(* IEC 61131-3 sources: verifaps-lib/share/oscat, 100 files *)

(* ---- 10_standard.st ---- *)
// Down Counter

PROGRAM standard
  VAR_INPUT
    input : INT;
  END_VAR
  VAR
    reset, cnt, max, init : INT;
  END_VAR

  ACTION act_Init
    cnt := max;
  END_ACTION

  ACTION act_Check
  END_ACTION

  ACTION act_Count
    cnt := cnt - 1;
  END_ACTION

  ACTION act_Reset
    cnt := max;
  END_ACTION

  ACTION act_End
  END_ACTION

  INITIAL_STEP Init
    : act_Init(N);
  END_STEP

  STEP Check
    : act_Check(N);
  END_STEP

  STEP Count
    : act_Count(N);
  END_STEP

  STEP Reset
    : act_Reset(N);
  END_STEP

  STEP End
    : act_End(N);
  END_STEP

  TRANSITION FROM Init TO Check
    := init;
  END_TRANSITION
  TRANSITION FROM Check TO Count
    := input == 1 and cnt > 0;
  END_TRANSITION
  TRANSITION FROM Count TO Check
    := True;
  END_TRANSITION
  TRANSITION FROM Check TO Reset
    := reset == 1;
  END_TRANSITION
  TRANSITION FROM Reset TO Check
    := True;
  END_TRANSITION
END_PROGRAM

(* ---- 10_upgraded.st ---- *)
// Down Counter (Upgraded)

PROGRAM upgraded
  VAR_INPUT
    input : INT;
  END_VAR
  VAR
    reset, cnt, max, init : INT;
  END_VAR

  ACTION act_Init
    cnt := max;
  END_ACTION

  ACTION act_Check
  END_ACTION

  ACTION act_Count
    cnt := cnt - 2;
  END_ACTION

  ACTION act_Reset
    cnt := max;
  END_ACTION

  ACTION act_End
  END_ACTION

  INITIAL_STEP Init
    : act_Init(N);
  END_STEP

  STEP Check
    : act_Check(N);
  END_STEP

  STEP Count
    : act_Count(N);
  END_STEP

  STEP Reset
    : act_Reset(N);
  END_STEP

  STEP End
    : act_End(N);
  END_STEP

  TRANSITION FROM Init TO Check
    := init;
  END_TRANSITION
  TRANSITION FROM Check TO Count
    := input == 1 and cnt > 0;
  END_TRANSITION
  TRANSITION FROM Count TO Check
    := True;
  END_TRANSITION
  TRANSITION FROM Check TO Reset
    := reset == 1;
  END_TRANSITION
  TRANSITION FROM Reset TO Check
    := True;
  END_TRANSITION
END_PROGRAM

(* ---- 11_standard.st ---- *)
// Comparator Greater

PROGRAM standard
  VAR
    a, b, out, init : INT;
  END_VAR

  ACTION act_Init
    out := 0;
  END_ACTION

  ACTION act_Check
  END_ACTION

  ACTION act_Set
    out := 1;
  END_ACTION

  ACTION act_Reset
    out := 0;
  END_ACTION

  ACTION act_End
  END_ACTION

  INITIAL_STEP Init
    : act_Init(N);
  END_STEP

  STEP Check
    : act_Check(N);
  END_STEP

  STEP Set
    : act_Set(N);
  END_STEP

  STEP Reset
    : act_Reset(N);
  END_STEP

  STEP End
    : act_End(N);
  END_STEP

  TRANSITION FROM Init TO Check
    := init;
  END_TRANSITION
  TRANSITION FROM Check TO Set
    := a > b;
  END_TRANSITION
  TRANSITION FROM Check TO Reset
    := a <= b;
  END_TRANSITION
  TRANSITION FROM Set TO End
    := True;
  END_TRANSITION
  TRANSITION FROM Reset TO End
    := True;
  END_TRANSITION
END_PROGRAM

(* ---- 11_upgraded.st ---- *)
// Comparator Greater (Upgraded)

PROGRAM upgraded
  VAR
    a, b, out, init : INT;
  END_VAR

  ACTION act_Init
    out := 0;
  END_ACTION

  ACTION act_Check
  END_ACTION

  ACTION act_Set
    out := a - b;
  END_ACTION

  ACTION act_Reset
    out := 0;
  END_ACTION

  ACTION act_End
  END_ACTION

  INITIAL_STEP Init
    : act_Init(N);
  END_STEP

  STEP Check
    : act_Check(N);
  END_STEP

  STEP Set
    : act_Set(N);
  END_STEP

  STEP Reset
    : act_Reset(N);
  END_STEP

  STEP End
    : act_End(N);
  END_STEP

  TRANSITION FROM Init TO Check
    := init;
  END_TRANSITION
  TRANSITION FROM Check TO Set
    := a > b;
  END_TRANSITION
  TRANSITION FROM Check TO Reset
    := a <= b;
  END_TRANSITION
  TRANSITION FROM Set TO End
    := True;
  END_TRANSITION
  TRANSITION FROM Reset TO End
    := True;
  END_TRANSITION
END_PROGRAM

(* ---- 12_standard.st ---- *)
// Comparator Less

PROGRAM standard
  VAR
    a, b, out, init : INT;
  END_VAR

  ACTION act_Init
    out := 0;
  END_ACTION

  ACTION act_Check
  END_ACTION

  ACTION act_Set
    out := 1;
  END_ACTION

  ACTION act_Reset
    out := 0;
  END_ACTION

  ACTION act_End
  END_ACTION

  INITIAL_STEP Init
    : act_Init(N);
  END_STEP

  STEP Check
    : act_Check(N);
  END_STEP

  STEP Set
    : act_Set(N);
  END_STEP

  STEP Reset
    : act_Reset(N);
  END_STEP

  STEP End
    : act_End(N);
  END_STEP

  TRANSITION FROM Init TO Check
    := init;
  END_TRANSITION
  TRANSITION FROM Check TO Set
    := a < b;
  END_TRANSITION
  TRANSITION FROM Check TO Reset
    := a >= b;
  END_TRANSITION
  TRANSITION FROM Set TO End
    := True;
  END_TRANSITION
  TRANSITION FROM Reset TO End
    := True;
  END_TRANSITION
END_PROGRAM

(* ---- 12_upgraded.st ---- *)
// Comparator Less (Upgraded)

PROGRAM upgraded
  VAR
    a, b, out, init : INT;
  END_VAR

  ACTION act_Init
    out := 0;
  END_ACTION

  ACTION act_Check
  END_ACTION

  ACTION act_Set
    out := b - a;
  END_ACTION

  ACTION act_Reset
    out := 0;
  END_ACTION

  ACTION act_End
  END_ACTION

  INITIAL_STEP Init
    : act_Init(N);
  END_STEP

  STEP Check
    : act_Check(N);
  END_STEP

  STEP Set
    : act_Set(N);
  END_STEP

  STEP Reset
    : act_Reset(N);
  END_STEP

  STEP End
    : act_End(N);
  END_STEP

  TRANSITION FROM Init TO Check
    := init;
  END_TRANSITION
  TRANSITION FROM Check TO Set
    := a < b;
  END_TRANSITION
  TRANSITION FROM Check TO Reset
    := a >= b;
  END_TRANSITION
  TRANSITION FROM Set TO End
    := True;
  END_TRANSITION
  TRANSITION FROM Reset TO End
    := True;
  END_TRANSITION
END_PROGRAM

(* ---- 13_standard.st ---- *)
// Comparator Equal

PROGRAM standard
  VAR
    a, b, out, init : INT;
  END_VAR

  ACTION act_Init
    out := 0;
  END_ACTION

  ACTION act_Check
  END_ACTION

  ACTION act_Set
    out := 1;
  END_ACTION

  ACTION act_Reset
    out := 0;
  END_ACTION

  ACTION act_End
  END_ACTION

  INITIAL_STEP Init
    : act_Init(N);
  END_STEP

  STEP Check
    : act_Check(N);
  END_STEP

  STEP Set
    : act_Set(N);
  END_STEP

  STEP Reset
    : act_Reset(N);
  END_STEP

  STEP End
    : act_End(N);
  END_STEP

  TRANSITION FROM Init TO Check
    := init;
  END_TRANSITION
  TRANSITION FROM Check TO Set
    := a == b;
  END_TRANSITION
  TRANSITION FROM Check TO Reset
    := a != b;
  END_TRANSITION
  TRANSITION FROM Set TO End
    := True;
  END_TRANSITION
  TRANSITION FROM Reset TO End
    := True;
  END_TRANSITION
END_PROGRAM

(* ---- 13_upgraded.st ---- *)
// Comparator Equal (Upgraded)

PROGRAM upgraded
  VAR
    a, b, out, init : INT;
  END_VAR

  ACTION act_Init
    out := 0;
  END_ACTION

  ACTION act_Check
  END_ACTION

  ACTION act_Set
    out := a + b;
  END_ACTION

  ACTION act_Reset
    out := 0;
  END_ACTION

  ACTION act_End
  END_ACTION

  INITIAL_STEP Init
    : act_Init(N);
  END_STEP

  STEP Check
    : act_Check(N);
  END_STEP

  STEP Set
    : act_Set(N);
  END_STEP

  STEP Reset
    : act_Reset(N);
  END_STEP

  STEP End
    : act_End(N);
  END_STEP

  TRANSITION FROM Init TO Check
    := init;
  END_TRANSITION
  TRANSITION FROM Check TO Set
    := a == b;
  END_TRANSITION
  TRANSITION FROM Check TO Reset
    := a != b;
  END_TRANSITION
  TRANSITION FROM Set TO End
    := True;
  END_TRANSITION
  TRANSITION FROM Reset TO End
    := True;
  END_TRANSITION
END_PROGRAM

(* ---- 14_standard.st ---- *)
// Comparator Not Equal

PROGRAM standard
  VAR
    a, b, out, init : INT;
  END_VAR

  ACTION act_Init
    out := 0;
  END_ACTION

  ACTION act_Check
  END_ACTION

  ACTION act_Set
    out := 1;
  END_ACTION

  ACTION act_Reset
    out := 0;
  END_ACTION

  ACTION act_End
  END_ACTION

  INITIAL_STEP Init
    : act_Init(N);
  END_STEP

  STEP Check
    : act_Check(N);
  END_STEP

  STEP Set
    : act_Set(N);
  END_STEP

  STEP Reset
    : act_Reset(N);
  END_STEP

  STEP End
    : act_End(N);
  END_STEP

  TRANSITION FROM Init TO Check
    := init;
  END_TRANSITION
  TRANSITION FROM Check TO Set
    := a != b;
  END_TRANSITION
  TRANSITION FROM Check TO Reset
    := a == b;
  END_TRANSITION
  TRANSITION FROM Set TO End
    := True;
  END_TRANSITION
  TRANSITION FROM Reset TO End
    := True;
  END_TRANSITION
END_PROGRAM

(* ---- 14_upgraded.st ---- *)
// Comparator Not Equal (Upgraded)

PROGRAM upgraded
  VAR
    a, b, out, init : INT;
  END_VAR

  ACTION act_Init
    out := 0;
  END_ACTION

  ACTION act_Check
  END_ACTION

  ACTION act_Set
    out := abs(a - b);
  END_ACTION

  ACTION act_Reset
    out := 0;
  END_ACTION

  ACTION act_End
  END_ACTION

  INITIAL_STEP Init
    : act_Init(N);
  END_STEP

  STEP Check
    : act_Check(N);
  END_STEP

  STEP Set
    : act_Set(N);
  END_STEP

  STEP Reset
    : act_Reset(N);
  END_STEP

  STEP End
    : act_End(N);
  END_STEP

  TRANSITION FROM Init TO Check
    := init;
  END_TRANSITION
  TRANSITION FROM Check TO Set
    := a != b;
  END_TRANSITION
  TRANSITION FROM Check TO Reset
    := a == b;
  END_TRANSITION
  TRANSITION FROM Set TO End
    := True;
  END_TRANSITION
  TRANSITION FROM Reset TO End
    := True;
  END_TRANSITION
END_PROGRAM

(* ---- 15_standard.st ---- *)
// Limit Upper Bound

PROGRAM standard
  VAR_INPUT
    input : INT;
  END_VAR
  VAR
    upper, out, init : INT;
  END_VAR

  ACTION act_Init
    out := input;
  END_ACTION

  ACTION act_Check
  END_ACTION

  ACTION act_Clamp
    out := upper;
  END_ACTION

  ACTION act_End
  END_ACTION

  INITIAL_STEP Init
    : act_Init(N);
  END_STEP

  STEP Check
    : act_Check(N);
  END_STEP

  STEP Clamp
    : act_Clamp(N);
  END_STEP

  STEP End
    : act_End(N);
  END_STEP

  TRANSITION FROM Init TO Check
    := init;
  END_TRANSITION
  TRANSITION FROM Check TO Clamp
    := input > upper;
  END_TRANSITION
  TRANSITION FROM Check TO End
    := input <= upper;
  END_TRANSITION
  TRANSITION FROM Clamp TO End
    := True;
  END_TRANSITION
END_PROGRAM

(* ---- 15_upgraded.st ---- *)
// Limit Upper Bound (Upgraded)

PROGRAM upgraded
  VAR_INPUT
    input : INT;
  END_VAR
  VAR
    upper, out, init : INT;
  END_VAR

  ACTION act_Init
    out := input + upper;
  END_ACTION

  ACTION act_Check
  END_ACTION

  ACTION act_Clamp
    out := upper;
  END_ACTION

  ACTION act_End
  END_ACTION

  INITIAL_STEP Init
    : act_Init(N);
  END_STEP

  STEP Check
    : act_Check(N);
  END_STEP

  STEP Clamp
    : act_Clamp(N);
  END_STEP

  STEP End
    : act_End(N);
  END_STEP

  TRANSITION FROM Init TO Check
    := init;
  END_TRANSITION
  TRANSITION FROM Check TO Clamp
    := input > upper;
  END_TRANSITION
  TRANSITION FROM Check TO End
    := input <= upper;
  END_TRANSITION
  TRANSITION FROM Clamp TO End
    := True;
  END_TRANSITION
END_PROGRAM

(* ---- 16_standard.st ---- *)
// Limit Lower Bound

PROGRAM standard
  VAR_INPUT
    input : INT;
  END_VAR
  VAR
    lower, out, init : INT;
  END_VAR

  ACTION act_Init
    out := input;
  END_ACTION

  ACTION act_Check
  END_ACTION

  ACTION act_Clamp
    out := lower;
  END_ACTION

  ACTION act_End
  END_ACTION

  INITIAL_STEP Init
    : act_Init(N);
  END_STEP

  STEP Check
    : act_Check(N);
  END_STEP

  STEP Clamp
    : act_Clamp(N);
  END_STEP

  STEP End
    : act_End(N);
  END_STEP

  TRANSITION FROM Init TO Check
    := init;
  END_TRANSITION
  TRANSITION FROM Check TO Clamp
    := input < lower;
  END_TRANSITION
  TRANSITION FROM Check TO End
    := input >= lower;
  END_TRANSITION
  TRANSITION FROM Clamp TO End
    := True;
  END_TRANSITION
END_PROGRAM

(* ---- 16_upgraded.st ---- *)
// Limit Lower Bound (Upgraded)

PROGRAM upgraded
  VAR_INPUT
    input : INT;
  END_VAR
  VAR
    lower, out, init : INT;
  END_VAR

  ACTION act_Init
    out := input - lower;
  END_ACTION

  ACTION act_Check
  END_ACTION

  ACTION act_Clamp
    out := lower;
  END_ACTION

  ACTION act_End
  END_ACTION

  INITIAL_STEP Init
    : act_Init(N);
  END_STEP

  STEP Check
    : act_Check(N);
  END_STEP

  STEP Clamp
    : act_Clamp(N);
  END_STEP

  STEP End
    : act_End(N);
  END_STEP

  TRANSITION FROM Init TO Check
    := init;
  END_TRANSITION
  TRANSITION FROM Check TO Clamp
    := input < lower;
  END_TRANSITION
  TRANSITION FROM Check TO End
    := input >= lower;
  END_TRANSITION
  TRANSITION FROM Clamp TO End
    := True;
  END_TRANSITION
END_PROGRAM

(* ---- 17_standard.st ---- *)
// Range Check

PROGRAM standard
  VAR_INPUT
    input : INT;
  END_VAR
  VAR
    low, high, in_range, init : INT;
  END_VAR

  ACTION act_Init
    in_range := 0;
  END_ACTION

  ACTION act_Check
  END_ACTION

  ACTION act_Set
    in_range := 1;
  END_ACTION

  ACTION act_Reset
    in_range := 0;
  END_ACTION

  ACTION act_End
  END_ACTION

  INITIAL_STEP Init
    : act_Init(N);
  END_STEP

  STEP Check
    : act_Check(N);
  END_STEP

  STEP Set
    : act_Set(N);
  END_STEP

  STEP Reset
    : act_Reset(N);
  END_STEP

  STEP End
    : act_End(N);
  END_STEP

  TRANSITION FROM Init TO Check
    := init;
  END_TRANSITION
  TRANSITION FROM Check TO Set
    := input >= low and input <= high;
  END_TRANSITION
  TRANSITION FROM Check TO Reset
    := input < low or input > high;
  END_TRANSITION
  TRANSITION FROM Set TO End
    := True;
  END_TRANSITION
  TRANSITION FROM Reset TO End
    := True;
  END_TRANSITION
END_PROGRAM

(* ---- 17_upgraded.st ---- *)
// Range Check (Upgraded)

PROGRAM upgraded
  VAR_INPUT
    input : INT;
  END_VAR
  VAR
    low, high, in_range, init : INT;
  END_VAR

  ACTION act_Init
    in_range := 0;
  END_ACTION

  ACTION act_Check
  END_ACTION

  ACTION act_Set
    in_range := input * 2;
  END_ACTION

  ACTION act_Reset
    in_range := input // 2;
  END_ACTION

  ACTION act_End
  END_ACTION

  INITIAL_STEP Init
    : act_Init(N);
  END_STEP

  STEP Check
    : act_Check(N);
  END_STEP

  STEP Set
    : act_Set(N);
  END_STEP

  STEP Reset
    : act_Reset(N);
  END_STEP

  STEP End
    : act_End(N);
  END_STEP

  TRANSITION FROM Init TO Check
    := init;
  END_TRANSITION
  TRANSITION FROM Check TO Set
    := input >= low and input <= high;
  END_TRANSITION
  TRANSITION FROM Check TO Reset
    := input < low or input > high;
  END_TRANSITION
  TRANSITION FROM Set TO End
    := True;
  END_TRANSITION
  TRANSITION FROM Reset TO End
    := True;
  END_TRANSITION
END_PROGRAM

(* ---- 18_standard.st ---- *)
// Rate Limiter (Ramp)

PROGRAM standard
  VAR_INPUT
    input : INT;
  END_VAR
  VAR
    out, rate, init : INT;
  END_VAR

  ACTION act_Init
    out := input;
  END_ACTION

  ACTION act_Check
  END_ACTION

  ACTION act_Inc
    out := out + rate;
  END_ACTION

  ACTION act_Dec
    out := out - rate;
  END_ACTION

  ACTION act_End
  END_ACTION

  INITIAL_STEP Init
    : act_Init(N);
  END_STEP

  STEP Check
    : act_Check(N);
  END_STEP

  STEP Inc
    : act_Inc(N);
  END_STEP

  STEP Dec
    : act_Dec(N);
  END_STEP

  STEP End
    : act_End(N);
  END_STEP

  TRANSITION FROM Init TO Check
    := init;
  END_TRANSITION
  TRANSITION FROM Check TO Inc
    := out < input;
  END_TRANSITION
  TRANSITION FROM Check TO Dec
    := out > input;
  END_TRANSITION
  TRANSITION FROM Check TO End
    := out == input;
  END_TRANSITION
  TRANSITION FROM Inc TO Check
    := True;
  END_TRANSITION
  TRANSITION FROM Dec TO Check
    := True;
  END_TRANSITION
END_PROGRAM

(* ---- 18_upgraded.st ---- *)
// Rate Limiter (Ramp) (Upgraded)

PROGRAM upgraded
  VAR_INPUT
    input : INT;
  END_VAR
  VAR
    out, rate, init : INT;
  END_VAR

  ACTION act_Init
    out := input;
  END_ACTION

  ACTION act_Check
  END_ACTION

  ACTION act_Inc
    out := out + 2*rate;
  END_ACTION

  ACTION act_Dec
    out := out - 2*rate;
  END_ACTION

  ACTION act_End
  END_ACTION

  INITIAL_STEP Init
    : act_Init(N);
  END_STEP

  STEP Check
    : act_Check(N);
  END_STEP

  STEP Inc
    : act_Inc(N);
  END_STEP

  STEP Dec
    : act_Dec(N);
  END_STEP

  STEP End
    : act_End(N);
  END_STEP

  TRANSITION FROM Init TO Check
    := init;
  END_TRANSITION
  TRANSITION FROM Check TO Inc
    := out < input;
  END_TRANSITION
  TRANSITION FROM Check TO Dec
    := out > input;
  END_TRANSITION
  TRANSITION FROM Check TO End
    := out == input;
  END_TRANSITION
  TRANSITION FROM Inc TO Check
    := True;
  END_TRANSITION
  TRANSITION FROM Dec TO Check
    := True;
  END_TRANSITION
END_PROGRAM

(* ---- 19_standard.st ---- *)
// Deadband

PROGRAM standard
  VAR_INPUT
    input : INT;
  END_VAR
  VAR
    upper, lower, out, init : INT;
  END_VAR

  ACTION act_Init
    out := 0;
  END_ACTION

  ACTION act_Check
  END_ACTION

  ACTION act_Pass
    out := input;
  END_ACTION

  ACTION act_Block
    out := 0;
  END_ACTION

  ACTION act_End
  END_ACTION

  INITIAL_STEP Init
    : act_Init(N);
  END_STEP

  STEP Check
    : act_Check(N);
  END_STEP

  STEP Pass
    : act_Pass(N);
  END_STEP

  STEP Block
    : act_Block(N);
  END_STEP

  STEP End
    : act_End(N);
  END_STEP

  TRANSITION FROM Init TO Check
    := init;
  END_TRANSITION
  TRANSITION FROM Check TO Pass
    := input > upper or input < lower;
  END_TRANSITION
  TRANSITION FROM Check TO Block
    := input <= upper and input >= lower;
  END_TRANSITION
  TRANSITION FROM Pass TO End
    := True;
  END_TRANSITION
  TRANSITION FROM Block TO End
    := True;
  END_TRANSITION
END_PROGRAM

(* ---- 19_upgraded.st ---- *)
// Deadband (Upgraded)

PROGRAM upgraded
  VAR_INPUT
    input : INT;
  END_VAR
  VAR
    upper, lower, out, init : INT;
  END_VAR

  ACTION act_Init
    out := 0;
  END_ACTION

  ACTION act_Check
  END_ACTION

  ACTION act_Pass
    out := input * 2;
  END_ACTION

  ACTION act_Block
    out := 0;
  END_ACTION

  ACTION act_End
  END_ACTION

  INITIAL_STEP Init
    : act_Init(N);
  END_STEP

  STEP Check
    : act_Check(N);
  END_STEP

  STEP Pass
    : act_Pass(N);
  END_STEP

  STEP Block
    : act_Block(N);
  END_STEP

  STEP End
    : act_End(N);
  END_STEP

  TRANSITION FROM Init TO Check
    := init;
  END_TRANSITION
  TRANSITION FROM Check TO Pass
    := input > upper or input < lower;
  END_TRANSITION
  TRANSITION FROM Check TO Block
    := input <= upper and input >= lower;
  END_TRANSITION
  TRANSITION FROM Pass TO End
    := True;
  END_TRANSITION
  TRANSITION FROM Block TO End
    := True;
  END_TRANSITION
END_PROGRAM

(* ---- 1_standard.st ---- *)
// Simple On-Off Control

PROGRAM standard
  VAR_INPUT
    input : INT;
  END_VAR
  VAR_OUTPUT
    output : INT;
  END_VAR
  VAR
    threshold, init : INT;
  END_VAR

  ACTION act_Init
    output := 0;
  END_ACTION

  ACTION act_Check
  END_ACTION

  ACTION act_On
    output := 1;
  END_ACTION

  ACTION act_Off
    output := 0;
  END_ACTION

  ACTION act_End
  END_ACTION

  INITIAL_STEP Init
    : act_Init(N);
  END_STEP

  STEP Check
    : act_Check(N);
  END_STEP

  STEP On
    : act_On(N);
  END_STEP

  STEP Off
    : act_Off(N);
  END_STEP

  STEP End
    : act_End(N);
  END_STEP

  TRANSITION FROM Init TO Check
    := init;
  END_TRANSITION
  TRANSITION FROM Check TO On
    := input > threshold;
  END_TRANSITION
  TRANSITION FROM Check TO Off
    := input <= threshold;
  END_TRANSITION
  TRANSITION FROM On TO End
    := True;
  END_TRANSITION
  TRANSITION FROM Off TO End
    := True;
  END_TRANSITION
END_PROGRAM

(* ---- 1_upgraded.st ---- *)
// Simple On-Off Control (Upgraded)

PROGRAM upgraded
  VAR_INPUT
    input : INT;
  END_VAR
  VAR_OUTPUT
    output : INT;
  END_VAR
  VAR
    threshold, gain, init : INT;
  END_VAR

  ACTION act_Init
    output := 0;
  END_ACTION

  ACTION act_Check
  END_ACTION

  ACTION act_On
    output := (input - threshold) * gain;
  END_ACTION

  ACTION act_Off
    output := 0;
  END_ACTION

  ACTION act_End
  END_ACTION

  INITIAL_STEP Init
    : act_Init(N);
  END_STEP

  STEP Check
    : act_Check(N);
  END_STEP

  STEP On
    : act_On(N);
  END_STEP

  STEP Off
    : act_Off(N);
  END_STEP

  STEP End
    : act_End(N);
  END_STEP

  TRANSITION FROM Init TO Check
    := init;
  END_TRANSITION
  TRANSITION FROM Check TO On
    := input > threshold;
  END_TRANSITION
  TRANSITION FROM Check TO Off
    := input <= threshold;
  END_TRANSITION
  TRANSITION FROM On TO End
    := True;
  END_TRANSITION
  TRANSITION FROM Off TO End
    := True;
  END_TRANSITION
END_PROGRAM

(* ---- 20_standard.st ---- *)
// Absolute Value

PROGRAM standard
  VAR_INPUT
    input : INT;
  END_VAR
  VAR
    out, init : INT;
  END_VAR

  ACTION act_Init
    out := input;
  END_ACTION

  ACTION act_Check
  END_ACTION

  ACTION act_Negate
    out := -input;
  END_ACTION

  ACTION act_End
  END_ACTION

  INITIAL_STEP Init
    : act_Init(N);
  END_STEP

  STEP Check
    : act_Check(N);
  END_STEP

  STEP Negate
    : act_Negate(N);
  END_STEP

  STEP End
    : act_End(N);
  END_STEP

  TRANSITION FROM Init TO Check
    := init;
  END_TRANSITION
  TRANSITION FROM Check TO Negate
    := input < 0;
  END_TRANSITION
  TRANSITION FROM Check TO End
    := input >= 0;
  END_TRANSITION
  TRANSITION FROM Negate TO End
    := True;
  END_TRANSITION
END_PROGRAM

(* ---- 20_upgraded.st ---- *)
// Absolute Value (Upgraded)

PROGRAM upgraded
  VAR_INPUT
    input : INT;
  END_VAR
  VAR
    out, init : INT;
  END_VAR

  ACTION act_Init
    out := abs(input);
  END_ACTION

  ACTION act_Check
  END_ACTION

  ACTION act_Negate
    out := -input;
  END_ACTION

  ACTION act_End
  END_ACTION

  INITIAL_STEP Init
    : act_Init(N);
  END_STEP

  STEP Check
    : act_Check(N);
  END_STEP

  STEP Negate
    : act_Negate(N);
  END_STEP

  STEP End
    : act_End(N);
  END_STEP

  TRANSITION FROM Init TO Check
    := init;
  END_TRANSITION
  TRANSITION FROM Check TO Negate
    := input < 0;
  END_TRANSITION
  TRANSITION FROM Check TO End
    := input >= 0;
  END_TRANSITION
  TRANSITION FROM Negate TO End
    := True;
  END_TRANSITION
END_PROGRAM

(* ---- 21_standard.st ---- *)
// Integrator

PROGRAM standard
  VAR_INPUT
    input : INT;
  END_VAR
  VAR
    enable, reset, sum, init : INT;
  END_VAR

  ACTION act_Init
    sum := 0;
  END_ACTION

  ACTION act_Check
  END_ACTION

  ACTION act_Add
    sum := sum + input;
  END_ACTION

  ACTION act_Reset
    sum := 0;
  END_ACTION

  ACTION act_End
  END_ACTION

  INITIAL_STEP Init
    : act_Init(N);
  END_STEP

  STEP Check
    : act_Check(N);
  END_STEP

  STEP Add
    : act_Add(N);
  END_STEP

  STEP Reset
    : act_Reset(N);
  END_STEP

  STEP End
    : act_End(N);
  END_STEP

  TRANSITION FROM Init TO Check
    := init;
  END_TRANSITION
  TRANSITION FROM Check TO Add
    := enable == 1;
  END_TRANSITION
  TRANSITION FROM Add TO Check
    := True;
  END_TRANSITION
  TRANSITION FROM Check TO Reset
    := reset == 1;
  END_TRANSITION
  TRANSITION FROM Reset TO Check
    := True;
  END_TRANSITION
END_PROGRAM

(* ---- 21_upgraded.st ---- *)
// Integrator (Upgraded)

PROGRAM upgraded
  VAR_INPUT
    input : INT;
  END_VAR
  VAR
    enable, reset, sum, init : INT;
  END_VAR

  ACTION act_Init
    sum := 0;
  END_ACTION

  ACTION act_Check
  END_ACTION

  ACTION act_Add
    sum := sum + input * 2;
  END_ACTION

  ACTION act_Reset
    sum := 0;
  END_ACTION

  ACTION act_End
  END_ACTION

  INITIAL_STEP Init
    : act_Init(N);
  END_STEP

  STEP Check
    : act_Check(N);
  END_STEP

  STEP Add
    : act_Add(N);
  END_STEP

  STEP Reset
    : act_Reset(N);
  END_STEP

  STEP End
    : act_End(N);
  END_STEP

  TRANSITION FROM Init TO Check
    := init;
  END_TRANSITION
  TRANSITION FROM Check TO Add
    := enable == 1;
  END_TRANSITION
  TRANSITION FROM Add TO Check
    := True;
  END_TRANSITION
  TRANSITION FROM Check TO Reset
    := reset == 1;
  END_TRANSITION
  TRANSITION FROM Reset TO Check
    := True;
  END_TRANSITION
END_PROGRAM

(* ---- 22_standard.st ---- *)
// Sample and Hold

PROGRAM standard
  VAR_INPUT
    input : INT;
  END_VAR
  VAR
    sample, hold, init : INT;
  END_VAR

  ACTION act_Init
    hold := 0;
  END_ACTION

  ACTION act_Check
  END_ACTION

  ACTION act_Sample
    hold := input;
  END_ACTION

  ACTION act_End
  END_ACTION

  INITIAL_STEP Init
    : act_Init(N);
  END_STEP

  STEP Check
    : act_Check(N);
  END_STEP

  STEP Sample
    : act_Sample(N);
  END_STEP

  STEP End
    : act_End(N);
  END_STEP

  TRANSITION FROM Init TO Check
    := init;
  END_TRANSITION
  TRANSITION FROM Check TO Sample
    := sample == 1;
  END_TRANSITION
  TRANSITION FROM Check TO End
    := sample == 0;
  END_TRANSITION
  TRANSITION FROM Sample TO End
    := True;
  END_TRANSITION
END_PROGRAM

(* ---- 22_upgraded.st ---- *)
// Sample and Hold (Upgraded)

PROGRAM upgraded
  VAR_INPUT
    input : INT;
  END_VAR
  VAR
    sample, hold, init : INT;
  END_VAR

  ACTION act_Init
    hold := 0;
  END_ACTION

  ACTION act_Check
  END_ACTION

  ACTION act_Sample
    hold := input + 1;
  END_ACTION

  ACTION act_End
  END_ACTION

  INITIAL_STEP Init
    : act_Init(N);
  END_STEP

  STEP Check
    : act_Check(N);
  END_STEP

  STEP Sample
    : act_Sample(N);
  END_STEP

  STEP End
    : act_End(N);
  END_STEP

  TRANSITION FROM Init TO Check
    := init;
  END_TRANSITION
  TRANSITION FROM Check TO Sample
    := sample == 1;
  END_TRANSITION
  TRANSITION FROM Check TO End
    := sample == 0;
  END_TRANSITION
  TRANSITION FROM Sample TO End
    := True;
  END_TRANSITION
END_PROGRAM

(* ---- 23_standard.st ---- *)
// S-R Latch

PROGRAM standard
  VAR
    s, r, q, init : INT;
  END_VAR

  ACTION act_Init
    q := 0;
  END_ACTION

  ACTION act_Check
  END_ACTION

  ACTION act_Set
    q := 1;
  END_ACTION

  ACTION act_Reset
    q := 0;
  END_ACTION

  ACTION act_End
  END_ACTION

  INITIAL_STEP Init
    : act_Init(N);
  END_STEP

  STEP Check
    : act_Check(N);
  END_STEP

  STEP Set
    : act_Set(N);
  END_STEP

  STEP Reset
    : act_Reset(N);
  END_STEP

  STEP End
    : act_End(N);
  END_STEP

  TRANSITION FROM Init TO Check
    := init;
  END_TRANSITION
  TRANSITION FROM Check TO Set
    := s == 1;
  END_TRANSITION
  TRANSITION FROM Check TO Reset
    := r == 1;
  END_TRANSITION
  TRANSITION FROM Set TO End
    := True;
  END_TRANSITION
  TRANSITION FROM Reset TO End
    := True;
  END_TRANSITION
END_PROGRAM

(* ---- 23_upgraded.st ---- *)
// S-R Latch (Upgraded)

PROGRAM upgraded
  VAR
    s, r, q, init : INT;
  END_VAR

  ACTION act_Init
    q := 0;
  END_ACTION

  ACTION act_Check
  END_ACTION

  ACTION act_Set
    q := 1;
  END_ACTION

  ACTION act_Reset
    q := -1;
  END_ACTION

  ACTION act_End
  END_ACTION

  INITIAL_STEP Init
    : act_Init(N);
  END_STEP

  STEP Check
    : act_Check(N);
  END_STEP

  STEP Set
    : act_Set(N);
  END_STEP

  STEP Reset
    : act_Reset(N);
  END_STEP

  STEP End
    : act_End(N);
  END_STEP

  TRANSITION FROM Init TO Check
    := init;
  END_TRANSITION
  TRANSITION FROM Check TO Set
    := s == 1;
  END_TRANSITION
  TRANSITION FROM Check TO Reset
    := r == 1;
  END_TRANSITION
  TRANSITION FROM Set TO End
    := True;
  END_TRANSITION
  TRANSITION FROM Reset TO End
    := True;
  END_TRANSITION
END_PROGRAM

(* ---- 24_standard.st ---- *)
// D Latch

PROGRAM standard
  VAR
    d, enable, q, init : INT;
  END_VAR

  ACTION act_Init
    q := 0;
  END_ACTION

  ACTION act_Check
  END_ACTION

  ACTION act_Latch
    q := d;
  END_ACTION

  ACTION act_End
  END_ACTION

  INITIAL_STEP Init
    : act_Init(N);
  END_STEP

  STEP Check
    : act_Check(N);
  END_STEP

  STEP Latch
    : act_Latch(N);
  END_STEP

  STEP End
    : act_End(N);
  END_STEP

  TRANSITION FROM Init TO Check
    := init;
  END_TRANSITION
  TRANSITION FROM Check TO Latch
    := enable == 1;
  END_TRANSITION
  TRANSITION FROM Check TO End
    := enable == 0;
  END_TRANSITION
  TRANSITION FROM Latch TO End
    := True;
  END_TRANSITION
END_PROGRAM

(* ---- 24_upgraded.st ---- *)
// D Latch (Upgraded)

PROGRAM upgraded
  VAR
    d, enable, q, init : INT;
  END_VAR

  ACTION act_Init
    q := 0;
  END_ACTION

  ACTION act_Check
  END_ACTION

  ACTION act_Latch
    q := d + 1;
  END_ACTION

  ACTION act_End
  END_ACTION

  INITIAL_STEP Init
    : act_Init(N);
  END_STEP

  STEP Check
    : act_Check(N);
  END_STEP

  STEP Latch
    : act_Latch(N);
  END_STEP

  STEP End
    : act_End(N);
  END_STEP

  TRANSITION FROM Init TO Check
    := init;
  END_TRANSITION
  TRANSITION FROM Check TO Latch
    := enable == 1;
  END_TRANSITION
  TRANSITION FROM Check TO End
    := enable == 0;
  END_TRANSITION
  TRANSITION FROM Latch TO End
    := True;
  END_TRANSITION
END_PROGRAM

(* ---- 25_standard.st ---- *)
// Up-Down Counter

PROGRAM standard
  VAR
    up, down, cnt, init : INT;
  END_VAR

  ACTION act_Init
    cnt := 0;
  END_ACTION

  ACTION act_Check
  END_ACTION

  ACTION act_Up
    cnt := cnt + 1;
  END_ACTION

  ACTION act_Down
    cnt := cnt - 1;
  END_ACTION

  ACTION act_End
  END_ACTION

  INITIAL_STEP Init
    : act_Init(N);
  END_STEP

  STEP Check
    : act_Check(N);
  END_STEP

  STEP Up
    : act_Up(N);
  END_STEP

  STEP Down
    : act_Down(N);
  END_STEP

  STEP End
    : act_End(N);
  END_STEP

  TRANSITION FROM Init TO Check
    := init;
  END_TRANSITION
  TRANSITION FROM Check TO Up
    := up == 1;
  END_TRANSITION
  TRANSITION FROM Check TO Down
    := down == 1;
  END_TRANSITION
  TRANSITION FROM Check TO End
    := up == 0 and down == 0;
  END_TRANSITION
  TRANSITION FROM Up TO End
    := True;
  END_TRANSITION
  TRANSITION FROM Down TO End
    := True;
  END_TRANSITION
END_PROGRAM

(* ---- 25_upgraded.st ---- *)
// Up-Down Counter (Upgraded)

PROGRAM upgraded
  VAR
    up, down, cnt, init : INT;
  END_VAR

  ACTION act_Init
    cnt := 0;
  END_ACTION

  ACTION act_Check
  END_ACTION

  ACTION act_Up
    cnt := cnt + 2;
  END_ACTION

  ACTION act_Down
    cnt := cnt - 2;
  END_ACTION

  ACTION act_End
  END_ACTION

  INITIAL_STEP Init
    : act_Init(N);
  END_STEP

  STEP Check
    : act_Check(N);
  END_STEP

  STEP Up
    : act_Up(N);
  END_STEP

  STEP Down
    : act_Down(N);
  END_STEP

  STEP End
    : act_End(N);
  END_STEP

  TRANSITION FROM Init TO Check
    := init;
  END_TRANSITION
  TRANSITION FROM Check TO Up
    := up == 1;
  END_TRANSITION
  TRANSITION FROM Check TO Down
    := down == 1;
  END_TRANSITION
  TRANSITION FROM Check TO End
    := up == 0 and down == 0;
  END_TRANSITION
  TRANSITION FROM Up TO End
    := True;
  END_TRANSITION
  TRANSITION FROM Down TO End
    := True;
  END_TRANSITION
END_PROGRAM

(* ---- 26_standard.st ---- *)
// Multiplexer (2-input)

PROGRAM standard
  VAR
    a, b, sel, out, init : INT;
  END_VAR

  ACTION act_Init
    out := a;
  END_ACTION

  ACTION act_Check
  END_ACTION

  ACTION act_SetB
    out := b;
  END_ACTION

  ACTION act_SetA
    out := a;
  END_ACTION

  ACTION act_End
  END_ACTION

  INITIAL_STEP Init
    : act_Init(N);
  END_STEP

  STEP Check
    : act_Check(N);
  END_STEP

  STEP SetB
    : act_SetB(N);
  END_STEP

  STEP SetA
    : act_SetA(N);
  END_STEP

  STEP End
    : act_End(N);
  END_STEP

  TRANSITION FROM Init TO Check
    := init;
  END_TRANSITION
  TRANSITION FROM Check TO SetB
    := sel == 1;
  END_TRANSITION
  TRANSITION FROM Check TO SetA
    := sel == 0;
  END_TRANSITION
  TRANSITION FROM SetB TO End
    := True;
  END_TRANSITION
  TRANSITION FROM SetA TO End
    := True;
  END_TRANSITION
END_PROGRAM

(* ---- 26_upgraded.st ---- *)
// Multiplexer (2-input) (Upgraded)

PROGRAM upgraded
  VAR
    a, b, sel, out, init : INT;
  END_VAR

  ACTION act_Init
    out := a + 1;
  END_ACTION

  ACTION act_Check
  END_ACTION

  ACTION act_SetB
    out := b + 1;
  END_ACTION

  ACTION act_SetA
    out := a + 1;
  END_ACTION

  ACTION act_End
  END_ACTION

  INITIAL_STEP Init
    : act_Init(N);
  END_STEP

  STEP Check
    : act_Check(N);
  END_STEP

  STEP SetB
    : act_SetB(N);
  END_STEP

  STEP SetA
    : act_SetA(N);
  END_STEP

  STEP End
    : act_End(N);
  END_STEP

  TRANSITION FROM Init TO Check
    := init;
  END_TRANSITION
  TRANSITION FROM Check TO SetB
    := sel == 1;
  END_TRANSITION
  TRANSITION FROM Check TO SetA
    := sel == 0;
  END_TRANSITION
  TRANSITION FROM SetB TO End
    := True;
  END_TRANSITION
  TRANSITION FROM SetA TO End
    := True;
  END_TRANSITION
END_PROGRAM

(* ---- 27_standard.st ---- *)
// Minimum Selector

PROGRAM standard
  VAR
    a, b, out, init : INT;
  END_VAR

  ACTION act_Init
    out := a;
  END_ACTION

  ACTION act_Check
  END_ACTION

  ACTION act_SetB
    out := b;
  END_ACTION

  ACTION act_End
  END_ACTION

  INITIAL_STEP Init
    : act_Init(N);
  END_STEP

  STEP Check
    : act_Check(N);
  END_STEP

  STEP SetB
    : act_SetB(N);
  END_STEP

  STEP End
    : act_End(N);
  END_STEP

  TRANSITION FROM Init TO Check
    := init;
  END_TRANSITION
  TRANSITION FROM Check TO SetB
    := b < a;
  END_TRANSITION
  TRANSITION FROM Check TO End
    := a <= b;
  END_TRANSITION
  TRANSITION FROM SetB TO End
    := True;
  END_TRANSITION
END_PROGRAM

(* ---- 27_upgraded.st ---- *)
// Minimum Selector (Upgraded)

PROGRAM upgraded
  VAR
    a, b, out, init : INT;
  END_VAR

  ACTION act_Init
    out := a - b;
  END_ACTION

  ACTION act_Check
  END_ACTION

  ACTION act_SetB
    out := b - a;
  END_ACTION

  ACTION act_End
  END_ACTION

  INITIAL_STEP Init
    : act_Init(N);
  END_STEP

  STEP Check
    : act_Check(N);
  END_STEP

  STEP SetB
    : act_SetB(N);
  END_STEP

  STEP End
    : act_End(N);
  END_STEP

  TRANSITION FROM Init TO Check
    := init;
  END_TRANSITION
  TRANSITION FROM Check TO SetB
    := b < a;
  END_TRANSITION
  TRANSITION FROM Check TO End
    := a <= b;
  END_TRANSITION
  TRANSITION FROM SetB TO End
    := True;
  END_TRANSITION
END_PROGRAM

(* ---- 28_standard.st ---- *)
// Maximum Selector

PROGRAM standard
  VAR
    a, b, out, init : INT;
  END_VAR

  ACTION act_Init
    out := a;
  END_ACTION

  ACTION act_Check
  END_ACTION

  ACTION act_SetB
    out := b;
  END_ACTION

  ACTION act_End
  END_ACTION

  INITIAL_STEP Init
    : act_Init(N);
  END_STEP

  STEP Check
    : act_Check(N);
  END_STEP

  STEP SetB
    : act_SetB(N);
  END_STEP

  STEP End
    : act_End(N);
  END_STEP

  TRANSITION FROM Init TO Check
    := init;
  END_TRANSITION
  TRANSITION FROM Check TO SetB
    := b > a;
  END_TRANSITION
  TRANSITION FROM Check TO End
    := a >= b;
  END_TRANSITION
  TRANSITION FROM SetB TO End
    := True;
  END_TRANSITION
END_PROGRAM

(* ---- 28_upgraded.st ---- *)
// Maximum Selector (Upgraded)

PROGRAM upgraded
  VAR
    a, b, out, init : INT;
  END_VAR

  ACTION act_Init
    out := a * 2;
  END_ACTION

  ACTION act_Check
  END_ACTION

  ACTION act_SetB
    out := b * 2;
  END_ACTION

  ACTION act_End
  END_ACTION

  INITIAL_STEP Init
    : act_Init(N);
  END_STEP

  STEP Check
    : act_Check(N);
  END_STEP

  STEP SetB
    : act_SetB(N);
  END_STEP

  STEP End
    : act_End(N);
  END_STEP

  TRANSITION FROM Init TO Check
    := init;
  END_TRANSITION
  TRANSITION FROM Check TO SetB
    := b > a;
  END_TRANSITION
  TRANSITION FROM Check TO End
    := a >= b;
  END_TRANSITION
  TRANSITION FROM SetB TO End
    := True;
  END_TRANSITION
END_PROGRAM

(* ---- 29_standard.st ---- *)
// Simple Arithmetic (a+b-c)

PROGRAM standard
  VAR
    a, b, c, out, init : INT;
  END_VAR

  ACTION act_Init
    out := a + b - c;
  END_ACTION

  ACTION act_End
  END_ACTION

  INITIAL_STEP Init
    : act_Init(N);
  END_STEP

  STEP End
    : act_End(N);
  END_STEP

  TRANSITION FROM Init TO End
    := init;
  END_TRANSITION
END_PROGRAM

(* ---- 29_upgraded.st ---- *)
// Simple Arithmetic (a+b-c) (Upgraded)

PROGRAM upgraded
  VAR
    a, b, c, out, init : INT;
  END_VAR

  ACTION act_Init
    out := a + b - c + 1;
  END_ACTION

  ACTION act_End
  END_ACTION

  INITIAL_STEP Init
    : act_Init(N);
  END_STEP

  STEP End
    : act_End(N);
  END_STEP

  TRANSITION FROM Init TO End
    := init;
  END_TRANSITION
END_PROGRAM

(* ---- 2_standard.st ---- *)
// Hysteresis Switch

PROGRAM standard
  VAR_INPUT
    input : INT;
  END_VAR
  VAR_OUTPUT
    output : INT;
  END_VAR
  VAR
    on_threshold, off_threshold, init : INT;
  END_VAR

  ACTION act_Init
    output := 0;
  END_ACTION

  ACTION act_Check
  END_ACTION

  ACTION act_On
    output := 1;
  END_ACTION

  ACTION act_Off
    output := 0;
  END_ACTION

  ACTION act_End
  END_ACTION

  INITIAL_STEP Init
    : act_Init(N);
  END_STEP

  STEP Check
    : act_Check(N);
  END_STEP

  STEP On
    : act_On(N);
  END_STEP

  STEP Off
    : act_Off(N);
  END_STEP

  STEP End
    : act_End(N);
  END_STEP

  TRANSITION FROM Init TO Check
    := init;
  END_TRANSITION
  TRANSITION FROM Check TO On
    := input > on_threshold;
  END_TRANSITION
  TRANSITION FROM Check TO Off
    := input < off_threshold;
  END_TRANSITION
  TRANSITION FROM On TO Check
    := True;
  END_TRANSITION
  TRANSITION FROM Off TO Check
    := True;
  END_TRANSITION
  TRANSITION FROM Check TO End
    := False;
  END_TRANSITION
END_PROGRAM

(* ---- 2_upgraded.st ---- *)
// Hysteresis Switch (Upgraded)

PROGRAM upgraded
  VAR_INPUT
    input : INT;
  END_VAR
  VAR_OUTPUT
    output : INT;
  END_VAR
  VAR
    on_threshold, off_threshold, scale, init : INT;
  END_VAR

  ACTION act_Init
    output := 0;
  END_ACTION

  ACTION act_Check
  END_ACTION

  ACTION act_On
    output := input * scale;
  END_ACTION

  ACTION act_Off
    output := 0;
  END_ACTION

  ACTION act_End
  END_ACTION

  INITIAL_STEP Init
    : act_Init(N);
  END_STEP

  STEP Check
    : act_Check(N);
  END_STEP

  STEP On
    : act_On(N);
  END_STEP

  STEP Off
    : act_Off(N);
  END_STEP

  STEP End
    : act_End(N);
  END_STEP

  TRANSITION FROM Init TO Check
    := init;
  END_TRANSITION
  TRANSITION FROM Check TO On
    := input > on_threshold;
  END_TRANSITION
  TRANSITION FROM Check TO Off
    := input < off_threshold;
  END_TRANSITION
  TRANSITION FROM On TO Check
    := True;
  END_TRANSITION
  TRANSITION FROM Off TO Check
    := True;
  END_TRANSITION
  TRANSITION FROM Check TO End
    := False;
  END_TRANSITION
END_PROGRAM

(* ---- 30_standard.st ---- *)
// Signum

PROGRAM standard
  VAR_INPUT
    input : INT;
  END_VAR
  VAR
    sgn, init : INT;
  END_VAR

  ACTION act_Init
    sgn := 0;
  END_ACTION

  ACTION act_Check
  END_ACTION

  ACTION act_SetPos
    sgn := 1;
  END_ACTION

  ACTION act_SetNeg
    sgn := -1;
  END_ACTION

  ACTION act_End
  END_ACTION

  INITIAL_STEP Init
    : act_Init(N);
  END_STEP

  STEP Check
    : act_Check(N);
  END_STEP

  STEP SetPos
    : act_SetPos(N);
  END_STEP

  STEP SetNeg
    : act_SetNeg(N);
  END_STEP

  STEP End
    : act_End(N);
  END_STEP

  TRANSITION FROM Init TO Check
    := init;
  END_TRANSITION
  TRANSITION FROM Check TO SetPos
    := input > 0;
  END_TRANSITION
  TRANSITION FROM Check TO SetNeg
    := input < 0;
  END_TRANSITION
  TRANSITION FROM Check TO End
    := input == 0;
  END_TRANSITION
  TRANSITION FROM SetPos TO End
    := True;
  END_TRANSITION
  TRANSITION FROM SetNeg TO End
    := True;
  END_TRANSITION
END_PROGRAM

(* ---- 30_upgraded.st ---- *)
// Signum (Upgraded)

PROGRAM upgraded
  VAR_INPUT
    input : INT;
  END_VAR
  VAR
    sgn, init : INT;
  END_VAR

  ACTION act_Init
    sgn := 0;
  END_ACTION

  ACTION act_Check
  END_ACTION

  ACTION act_SetPos
    sgn := input;
  END_ACTION

  ACTION act_SetNeg
    sgn := -input;
  END_ACTION

  ACTION act_End
  END_ACTION

  INITIAL_STEP Init
    : act_Init(N);
  END_STEP

  STEP Check
    : act_Check(N);
  END_STEP

  STEP SetPos
    : act_SetPos(N);
  END_STEP

  STEP SetNeg
    : act_SetNeg(N);
  END_STEP

  STEP End
    : act_End(N);
  END_STEP

  TRANSITION FROM Init TO Check
    := init;
  END_TRANSITION
  TRANSITION FROM Check TO SetPos
    := input > 0;
  END_TRANSITION
  TRANSITION FROM Check TO SetNeg
    := input < 0;
  END_TRANSITION
  TRANSITION FROM Check TO End
    := input == 0;
  END_TRANSITION
  TRANSITION FROM SetPos TO End
    := True;
  END_TRANSITION
  TRANSITION FROM SetNeg TO End
    := True;
  END_TRANSITION
END_PROGRAM

(* ---- 31_standard.st ---- *)
// Increment If

PROGRAM standard
  VAR
    cond, count, init : INT;
  END_VAR

  ACTION act_Init
    count := 0;
  END_ACTION

  ACTION act_Check
  END_ACTION

  ACTION act_Inc
    count := count + 1;
  END_ACTION

  ACTION act_End
  END_ACTION

  INITIAL_STEP Init
    : act_Init(N);
  END_STEP

  STEP Check
    : act_Check(N);
  END_STEP

  STEP Inc
    : act_Inc(N);
  END_STEP

  STEP End
    : act_End(N);
  END_STEP

  TRANSITION FROM Init TO Check
    := init;
  END_TRANSITION
  TRANSITION FROM Check TO Inc
    := cond == 1;
  END_TRANSITION
  TRANSITION FROM Check TO End
    := cond == 0;
  END_TRANSITION
  TRANSITION FROM Inc TO End
    := True;
  END_TRANSITION
END_PROGRAM

(* ---- 31_upgraded.st ---- *)
// Increment If (Upgraded)

PROGRAM upgraded
  VAR
    cond, count, init : INT;
  END_VAR

  ACTION act_Init
    count := 0;
  END_ACTION

  ACTION act_Check
  END_ACTION

  ACTION act_Inc
    count := count + 2;
  END_ACTION

  ACTION act_End
  END_ACTION

  INITIAL_STEP Init
    : act_Init(N);
  END_STEP

  STEP Check
    : act_Check(N);
  END_STEP

  STEP Inc
    : act_Inc(N);
  END_STEP

  STEP End
    : act_End(N);
  END_STEP

  TRANSITION FROM Init TO Check
    := init;
  END_TRANSITION
  TRANSITION FROM Check TO Inc
    := cond == 1;
  END_TRANSITION
  TRANSITION FROM Check TO End
    := cond == 0;
  END_TRANSITION
  TRANSITION FROM Inc TO End
    := True;
  END_TRANSITION
END_PROGRAM

(* ---- 32_standard.st ---- *)
// Decrement If

PROGRAM standard
  VAR
    cond, count, init : INT;
  END_VAR

  ACTION act_Init
    count := 0;
  END_ACTION

  ACTION act_Check
  END_ACTION

  ACTION act_Dec
    count := count - 1;
  END_ACTION

  ACTION act_End
  END_ACTION

  INITIAL_STEP Init
    : act_Init(N);
  END_STEP

  STEP Check
    : act_Check(N);
  END_STEP

  STEP Dec
    : act_Dec(N);
  END_STEP

  STEP End
    : act_End(N);
  END_STEP

  TRANSITION FROM Init TO Check
    := init;
  END_TRANSITION
  TRANSITION FROM Check TO Dec
    := cond == 1;
  END_TRANSITION
  TRANSITION FROM Check TO End
    := cond == 0;
  END_TRANSITION
  TRANSITION FROM Dec TO End
    := True;
  END_TRANSITION
END_PROGRAM

(* ---- 32_upgraded.st ---- *)
// Decrement If (Upgraded)

PROGRAM upgraded
  VAR
    cond, count, init : INT;
  END_VAR

  ACTION act_Init
    count := 0;
  END_ACTION

  ACTION act_Check
  END_ACTION

  ACTION act_Dec
    count := count - 2;
  END_ACTION

  ACTION act_End
  END_ACTION

  INITIAL_STEP Init
    : act_Init(N);
  END_STEP

  STEP Check
    : act_Check(N);
  END_STEP

  STEP Dec
    : act_Dec(N);
  END_STEP

  STEP End
    : act_End(N);
  END_STEP

  TRANSITION FROM Init TO Check
    := init;
  END_TRANSITION
  TRANSITION FROM Check TO Dec
    := cond == 1;
  END_TRANSITION
  TRANSITION FROM Check TO End
    := cond == 0;
  END_TRANSITION
  TRANSITION FROM Dec TO End
    := True;
  END_TRANSITION
END_PROGRAM

(* ---- 33_standard.st ---- *)
// Clamp in Range

PROGRAM standard
  VAR_INPUT
    input : INT;
  END_VAR
  VAR
    low, high, out, init : INT;
  END_VAR

  ACTION act_Init
    out := input;
  END_ACTION

  ACTION act_Check
  END_ACTION

  ACTION act_ClampLow
    out := low;
  END_ACTION

  ACTION act_ClampHigh
    out := high;
  END_ACTION

  ACTION act_End
  END_ACTION

  INITIAL_STEP Init
    : act_Init(N);
  END_STEP

  STEP Check
    : act_Check(N);
  END_STEP

  STEP ClampLow
    : act_ClampLow(N);
  END_STEP

  STEP ClampHigh
    : act_ClampHigh(N);
  END_STEP

  STEP End
    : act_End(N);
  END_STEP

  TRANSITION FROM Init TO Check
    := init;
  END_TRANSITION
  TRANSITION FROM Check TO ClampLow
    := input < low;
  END_TRANSITION
  TRANSITION FROM Check TO ClampHigh
    := input > high;
  END_TRANSITION
  TRANSITION FROM Check TO End
    := input >= low and input <= high;
  END_TRANSITION
  TRANSITION FROM ClampLow TO End
    := True;
  END_TRANSITION
  TRANSITION FROM ClampHigh TO End
    := True;
  END_TRANSITION
END_PROGRAM

(* ---- 33_upgraded.st ---- *)
// Clamp in Range (Upgraded)

PROGRAM upgraded
  VAR_INPUT
    input : INT;
  END_VAR
  VAR
    low, high, out, init : INT;
  END_VAR

  ACTION act_Init
    out := input * 2;
  END_ACTION

  ACTION act_Check
  END_ACTION

  ACTION act_ClampLow
    out := low;
  END_ACTION

  ACTION act_ClampHigh
    out := high;
  END_ACTION

  ACTION act_End
  END_ACTION

  INITIAL_STEP Init
    : act_Init(N);
  END_STEP

  STEP Check
    : act_Check(N);
  END_STEP

  STEP ClampLow
    : act_ClampLow(N);
  END_STEP

  STEP ClampHigh
    : act_ClampHigh(N);
  END_STEP

  STEP End
    : act_End(N);
  END_STEP

  TRANSITION FROM Init TO Check
    := init;
  END_TRANSITION
  TRANSITION FROM Check TO ClampLow
    := input < low;
  END_TRANSITION
  TRANSITION FROM Check TO ClampHigh
    := input > high;
  END_TRANSITION
  TRANSITION FROM Check TO End
    := input >= low and input <= high;
  END_TRANSITION
  TRANSITION FROM ClampLow TO End
    := True;
  END_TRANSITION
  TRANSITION FROM ClampHigh TO End
    := True;
  END_TRANSITION
END_PROGRAM

(* ---- 34_standard.st ---- *)
// Invert

PROGRAM standard
  VAR_INPUT
    input : INT;
  END_VAR
  VAR
    out, init : INT;
  END_VAR

  ACTION act_Init
    out := -input;
  END_ACTION

  ACTION act_End
  END_ACTION

  INITIAL_STEP Init
    : act_Init(N);
  END_STEP

  STEP End
    : act_End(N);
  END_STEP

  TRANSITION FROM Init TO End
    := init;
  END_TRANSITION
END_PROGRAM

(* ---- 34_upgraded.st ---- *)
// Invert (Upgraded)

PROGRAM upgraded
  VAR_INPUT
    input : INT;
  END_VAR
  VAR
    out, init : INT;
  END_VAR

  ACTION act_Init
    out := -input * 2;
  END_ACTION

  ACTION act_End
  END_ACTION

  INITIAL_STEP Init
    : act_Init(N);
  END_STEP

  STEP End
    : act_End(N);
  END_STEP

  TRANSITION FROM Init TO End
    := init;
  END_TRANSITION
END_PROGRAM

(* ---- 35_standard.st ---- *)
// Resettable Counter

PROGRAM standard
  VAR
    enable, reset, count, init : INT;
  END_VAR

  ACTION act_Init
    count := 0;
  END_ACTION

  ACTION act_Check
  END_ACTION

  ACTION act_Inc
    count := count + 1;
  END_ACTION

  ACTION act_Reset
    count := 0;
  END_ACTION

  ACTION act_End
  END_ACTION

  INITIAL_STEP Init
    : act_Init(N);
  END_STEP

  STEP Check
    : act_Check(N);
  END_STEP

  STEP Inc
    : act_Inc(N);
  END_STEP

  STEP Reset
    : act_Reset(N);
  END_STEP

  STEP End
    : act_End(N);
  END_STEP

  TRANSITION FROM Init TO Check
    := init;
  END_TRANSITION
  TRANSITION FROM Check TO Inc
    := enable == 1;
  END_TRANSITION
  TRANSITION FROM Check TO Reset
    := reset == 1;
  END_TRANSITION
  TRANSITION FROM Inc TO End
    := True;
  END_TRANSITION
  TRANSITION FROM Reset TO End
    := True;
  END_TRANSITION
END_PROGRAM

(* ---- 35_upgraded.st ---- *)
// Resettable Counter (Upgraded)

PROGRAM upgraded
  VAR
    enable, reset, count, init : INT;
  END_VAR

  ACTION act_Init
    count := 0;
  END_ACTION

  ACTION act_Check
  END_ACTION

  ACTION act_Inc
    count := count + 3;
  END_ACTION

  ACTION act_Reset
    count := 0;
  END_ACTION

  ACTION act_End
  END_ACTION

  INITIAL_STEP Init
    : act_Init(N);
  END_STEP

  STEP Check
    : act_Check(N);
  END_STEP

  STEP Inc
    : act_Inc(N);
  END_STEP

  STEP Reset
    : act_Reset(N);
  END_STEP

  STEP End
    : act_End(N);
  END_STEP

  TRANSITION FROM Init TO Check
    := init;
  END_TRANSITION
  TRANSITION FROM Check TO Inc
    := enable == 1;
  END_TRANSITION
  TRANSITION FROM Check TO Reset
    := reset == 1;
  END_TRANSITION
  TRANSITION FROM Inc TO End
    := True;
  END_TRANSITION
  TRANSITION FROM Reset TO End
    := True;
  END_TRANSITION
END_PROGRAM

(* ---- 36_standard.st ---- *)
// Modulo Counter

PROGRAM standard
  VAR
    enable, mod, count, init : INT;
  END_VAR

  ACTION act_Init
    count := 0;
  END_ACTION

  ACTION act_Check
  END_ACTION

  ACTION act_Inc
    count := (count + 1) % mod;
  END_ACTION

  ACTION act_End
  END_ACTION

  INITIAL_STEP Init
    : act_Init(N);
  END_STEP

  STEP Check
    : act_Check(N);
  END_STEP

  STEP Inc
    : act_Inc(N);
  END_STEP

  STEP End
    : act_End(N);
  END_STEP

  TRANSITION FROM Init TO Check
    := init;
  END_TRANSITION
  TRANSITION FROM Check TO Inc
    := enable == 1;
  END_TRANSITION
  TRANSITION FROM Check TO End
    := enable == 0;
  END_TRANSITION
  TRANSITION FROM Inc TO End
    := True;
  END_TRANSITION
END_PROGRAM

(* ---- 36_upgraded.st ---- *)
// Modulo Counter (Upgraded)

PROGRAM upgraded
  VAR
    enable, mod, count, init : INT;
  END_VAR

  ACTION act_Init
    count := 0;
  END_ACTION

  ACTION act_Check
  END_ACTION

  ACTION act_Inc
    count := (count + 2) % mod;
  END_ACTION

  ACTION act_End
  END_ACTION

  INITIAL_STEP Init
    : act_Init(N);
  END_STEP

  STEP Check
    : act_Check(N);
  END_STEP

  STEP Inc
    : act_Inc(N);
  END_STEP

  STEP End
    : act_End(N);
  END_STEP

  TRANSITION FROM Init TO Check
    := init;
  END_TRANSITION
  TRANSITION FROM Check TO Inc
    := enable == 1;
  END_TRANSITION
  TRANSITION FROM Check TO End
    := enable == 0;
  END_TRANSITION
  TRANSITION FROM Inc TO End
    := True;
  END_TRANSITION
END_PROGRAM

(* ---- 37_standard.st ---- *)
// Comparator GE (>=)

PROGRAM standard
  VAR
    a, b, out, init : INT;
  END_VAR

  ACTION act_Init
    out := 0;
  END_ACTION

  ACTION act_Check
  END_ACTION

  ACTION act_Set
    out := 1;
  END_ACTION

  ACTION act_Reset
    out := 0;
  END_ACTION

  ACTION act_End
  END_ACTION

  INITIAL_STEP Init
    : act_Init(N);
  END_STEP

  STEP Check
    : act_Check(N);
  END_STEP

  STEP Set
    : act_Set(N);
  END_STEP

  STEP Reset
    : act_Reset(N);
  END_STEP

  STEP End
    : act_End(N);
  END_STEP

  TRANSITION FROM Init TO Check
    := init;
  END_TRANSITION
  TRANSITION FROM Check TO Set
    := a >= b;
  END_TRANSITION
  TRANSITION FROM Check TO Reset
    := a < b;
  END_TRANSITION
  TRANSITION FROM Set TO End
    := True;
  END_TRANSITION
  TRANSITION FROM Reset TO End
    := True;
  END_TRANSITION
END_PROGRAM

(* ---- 37_upgraded.st ---- *)
// Comparator GE (>=) (Upgraded)

PROGRAM upgraded
  VAR
    a, b, out, init : INT;
  END_VAR

  ACTION act_Init
    out := 0;
  END_ACTION

  ACTION act_Check
  END_ACTION

  ACTION act_Set
    out := a + b;
  END_ACTION

  ACTION act_Reset
    out := 0;
  END_ACTION

  ACTION act_End
  END_ACTION

  INITIAL_STEP Init
    : act_Init(N);
  END_STEP

  STEP Check
    : act_Check(N);
  END_STEP

  STEP Set
    : act_Set(N);
  END_STEP

  STEP Reset
    : act_Reset(N);
  END_STEP

  STEP End
    : act_End(N);
  END_STEP

  TRANSITION FROM Init TO Check
    := init;
  END_TRANSITION
  TRANSITION FROM Check TO Set
    := a >= b;
  END_TRANSITION
  TRANSITION FROM Check TO Reset
    := a < b;
  END_TRANSITION
  TRANSITION FROM Set TO End
    := True;
  END_TRANSITION
  TRANSITION FROM Reset TO End
    := True;
  END_TRANSITION
END_PROGRAM

(* ---- 38_standard.st ---- *)
// Comparator LE (<=)

PROGRAM standard
  VAR
    a, b, out, init : INT;
  END_VAR

  ACTION act_Init
    out := 0;
  END_ACTION

  ACTION act_Check
  END_ACTION

  ACTION act_Set
    out := 1;
  END_ACTION

  ACTION act_Reset
    out := 0;
  END_ACTION

  ACTION act_End
  END_ACTION

  INITIAL_STEP Init
    : act_Init(N);
  END_STEP

  STEP Check
    : act_Check(N);
  END_STEP

  STEP Set
    : act_Set(N);
  END_STEP

  STEP Reset
    : act_Reset(N);
  END_STEP

  STEP End
    : act_End(N);
  END_STEP

  TRANSITION FROM Init TO Check
    := init;
  END_TRANSITION
  TRANSITION FROM Check TO Set
    := a <= b;
  END_TRANSITION
  TRANSITION FROM Check TO Reset
    := a > b;
  END_TRANSITION
  TRANSITION FROM Set TO End
    := True;
  END_TRANSITION
  TRANSITION FROM Reset TO End
    := True;
  END_TRANSITION
END_PROGRAM

(* ---- 38_upgraded.st ---- *)
// Comparator LE (<=) (Upgraded)

PROGRAM upgraded
  VAR
    a, b, out, init : INT;
  END_VAR

  ACTION act_Init
    out := 0;
  END_ACTION

  ACTION act_Check
  END_ACTION

  ACTION act_Set
    out := a * b;
  END_ACTION

  ACTION act_Reset
    out := 0;
  END_ACTION

  ACTION act_End
  END_ACTION

  INITIAL_STEP Init
    : act_Init(N);
  END_STEP

  STEP Check
    : act_Check(N);
  END_STEP

  STEP Set
    : act_Set(N);
  END_STEP

  STEP Reset
    : act_Reset(N);
  END_STEP

  STEP End
    : act_End(N);
  END_STEP

  TRANSITION FROM Init TO Check
    := init;
  END_TRANSITION
  TRANSITION FROM Check TO Set
    := a <= b;
  END_TRANSITION
  TRANSITION FROM Check TO Reset
    := a > b;
  END_TRANSITION
  TRANSITION FROM Set TO End
    := True;
  END_TRANSITION
  TRANSITION FROM Reset TO End
    := True;
  END_TRANSITION
END_PROGRAM

(* ---- 39_standard.st ---- *)
// Set-Reset Flip-Flop (priority to set)

PROGRAM standard
  VAR
    set, reset, q, init : INT;
  END_VAR

  ACTION act_Init
    q := 0;
  END_ACTION

  ACTION act_Check
  END_ACTION

  ACTION act_Set
    q := 1;
  END_ACTION

  ACTION act_Reset
    q := 0;
  END_ACTION

  ACTION act_End
  END_ACTION

  INITIAL_STEP Init
    : act_Init(N);
  END_STEP

  STEP Check
    : act_Check(N);
  END_STEP

  STEP Set
    : act_Set(N);
  END_STEP

  STEP Reset
    : act_Reset(N);
  END_STEP

  STEP End
    : act_End(N);
  END_STEP

  TRANSITION FROM Init TO Check
    := init;
  END_TRANSITION
  TRANSITION FROM Check TO Set
    := set == 1;
  END_TRANSITION
  TRANSITION FROM Check TO Reset
    := reset == 1 and set == 0;
  END_TRANSITION
  TRANSITION FROM Check TO End
    := set == 0 and reset == 0;
  END_TRANSITION
  TRANSITION FROM Set TO End
    := True;
  END_TRANSITION
  TRANSITION FROM Reset TO End
    := True;
  END_TRANSITION
END_PROGRAM

(* ---- 39_upgraded.st ---- *)
// Set-Reset Flip-Flop (priority to set) (Upgraded)

PROGRAM upgraded
  VAR
    set, reset, q, init : INT;
  END_VAR

  ACTION act_Init
    q := 0;
  END_ACTION

  ACTION act_Check
  END_ACTION

  ACTION act_Set
    q := set + 1;
  END_ACTION

  ACTION act_Reset
    q := reset - 1;
  END_ACTION

  ACTION act_End
  END_ACTION

  INITIAL_STEP Init
    : act_Init(N);
  END_STEP

  STEP Check
    : act_Check(N);
  END_STEP

  STEP Set
    : act_Set(N);
  END_STEP

  STEP Reset
    : act_Reset(N);
  END_STEP

  STEP End
    : act_End(N);
  END_STEP

  TRANSITION FROM Init TO Check
    := init;
  END_TRANSITION
  TRANSITION FROM Check TO Set
    := set == 1;
  END_TRANSITION
  TRANSITION FROM Check TO Reset
    := reset == 1 and set == 0;
  END_TRANSITION
  TRANSITION FROM Check TO End
    := set == 0 and reset == 0;
  END_TRANSITION
  TRANSITION FROM Set TO End
    := True;
  END_TRANSITION
  TRANSITION FROM Reset TO End
    := True;
  END_TRANSITION
END_PROGRAM

(* ---- 3_standard.st ---- *)
// Toggle by Rising Edge (T Flip-Flop)

PROGRAM standard
  VAR_INPUT
    input : INT;
  END_VAR
  VAR_OUTPUT
    output : INT;
  END_VAR
  VAR
    last, init : INT;
  END_VAR

  ACTION act_Init
    output := 0; last := 0;
  END_ACTION

  ACTION act_Check
  END_ACTION

  ACTION act_Toggle
    output := 1 - output;
  END_ACTION

  ACTION act_End
    last := input;
  END_ACTION

  INITIAL_STEP Init
    : act_Init(N);
  END_STEP

  STEP Check
    : act_Check(N);
  END_STEP

  STEP Toggle
    : act_Toggle(N);
  END_STEP

  STEP End
    : act_End(N);
  END_STEP

  TRANSITION FROM Init TO Check
    := init;
  END_TRANSITION
  TRANSITION FROM Check TO Toggle
    := input == 1 and last == 0;
  END_TRANSITION
  TRANSITION FROM Toggle TO End
    := True;
  END_TRANSITION
  TRANSITION FROM Check TO End
    := input == 0 or last == 1;
  END_TRANSITION
END_PROGRAM

(* ---- 3_upgraded.st ---- *)
// Toggle by Rising Edge (T Flip-Flop) (Upgraded)

PROGRAM upgraded
  VAR_INPUT
    input : INT;
  END_VAR
  VAR_OUTPUT
    output : INT;
  END_VAR
  VAR
    last, toggle_count, init : INT;
  END_VAR

  ACTION act_Init
    output := 0; last := 0;
    toggle_count := 0;
  END_ACTION

  ACTION act_Check
  END_ACTION

  ACTION act_Toggle
    output := 1 - output;
    toggle_count := toggle_count + 1;
  END_ACTION

  ACTION act_End
    last := input;
  END_ACTION

  INITIAL_STEP Init
    : act_Init(N);
  END_STEP

  STEP Check
    : act_Check(N);
  END_STEP

  STEP Toggle
    : act_Toggle(N);
  END_STEP

  STEP End
    : act_End(N);
  END_STEP

  TRANSITION FROM Init TO Check
    := init;
  END_TRANSITION
  TRANSITION FROM Check TO Toggle
    := input == 1 and last == 0;
  END_TRANSITION
  TRANSITION FROM Toggle TO End
    := True;
  END_TRANSITION
  TRANSITION FROM Check TO End
    := input == 0 or last == 1;
  END_TRANSITION
END_PROGRAM

(* ---- 40_standard.st ---- *)
// Hold Last Value

PROGRAM standard
  VAR_INPUT
    input : INT;
  END_VAR
  VAR
    enable, hold, init : INT;
  END_VAR

  ACTION act_Init
    hold := 0;
  END_ACTION

  ACTION act_Check
  END_ACTION

  ACTION act_Hold
    hold := input;
  END_ACTION

  ACTION act_End
  END_ACTION

  INITIAL_STEP Init
    : act_Init(N);
  END_STEP

  STEP Check
    : act_Check(N);
  END_STEP

  STEP Hold
    : act_Hold(N);
  END_STEP

  STEP End
    : act_End(N);
  END_STEP

  TRANSITION FROM Init TO Check
    := init;
  END_TRANSITION
  TRANSITION FROM Check TO Hold
    := enable == 1;
  END_TRANSITION
  TRANSITION FROM Check TO End
    := enable == 0;
  END_TRANSITION
  TRANSITION FROM Hold TO End
    := True;
  END_TRANSITION
END_PROGRAM

(* ---- 40_upgraded.st ---- *)
// Hold Last Value (Upgraded)

PROGRAM upgraded
  VAR_INPUT
    input : INT;
  END_VAR
  VAR
    enable, hold, init : INT;
  END_VAR

  ACTION act_Init
    hold := 0;
  END_ACTION

  ACTION act_Check
  END_ACTION

  ACTION act_Hold
    hold := input + 2;
  END_ACTION

  ACTION act_End
  END_ACTION

  INITIAL_STEP Init
    : act_Init(N);
  END_STEP

  STEP Check
    : act_Check(N);
  END_STEP

  STEP Hold
    : act_Hold(N);
  END_STEP

  STEP End
    : act_End(N);
  END_STEP

  TRANSITION FROM Init TO Check
    := init;
  END_TRANSITION
  TRANSITION FROM Check TO Hold
    := enable == 1;
  END_TRANSITION
  TRANSITION FROM Check TO End
    := enable == 0;
  END_TRANSITION
  TRANSITION FROM Hold TO End
    := True;
  END_TRANSITION
END_PROGRAM

(* ---- 41_standard.st ---- *)
// Latch Until Reset

PROGRAM standard
  VAR
    set, reset, q, init : INT;
  END_VAR

  ACTION act_Init
    q := 0;
  END_ACTION

  ACTION act_Check
  END_ACTION

  ACTION act_Latch
    q := 1;
  END_ACTION

  ACTION act_Reset
    q := 0;
  END_ACTION

  ACTION act_End
  END_ACTION

  INITIAL_STEP Init
    : act_Init(N);
  END_STEP

  STEP Check
    : act_Check(N);
  END_STEP

  STEP Latch
    : act_Latch(N);
  END_STEP

  STEP Reset
    : act_Reset(N);
  END_STEP

  STEP End
    : act_End(N);
  END_STEP

  TRANSITION FROM Init TO Check
    := init;
  END_TRANSITION
  TRANSITION FROM Check TO Latch
    := set == 1;
  END_TRANSITION
  TRANSITION FROM Check TO Reset
    := reset == 1;
  END_TRANSITION
  TRANSITION FROM Check TO End
    := set == 0 and reset == 0;
  END_TRANSITION
  TRANSITION FROM Latch TO End
    := True;
  END_TRANSITION
  TRANSITION FROM Reset TO End
    := True;
  END_TRANSITION
END_PROGRAM

(* ---- 41_upgraded.st ---- *)
// Latch Until Reset (Upgraded)

PROGRAM upgraded
  VAR
    set, reset, q, init : INT;
  END_VAR

  ACTION act_Init
    q := 0;
  END_ACTION

  ACTION act_Check
  END_ACTION

  ACTION act_Latch
    q := set * 2;
  END_ACTION

  ACTION act_Reset
    q := reset * -1;
  END_ACTION

  ACTION act_End
  END_ACTION

  INITIAL_STEP Init
    : act_Init(N);
  END_STEP

  STEP Check
    : act_Check(N);
  END_STEP

  STEP Latch
    : act_Latch(N);
  END_STEP

  STEP Reset
    : act_Reset(N);
  END_STEP

  STEP End
    : act_End(N);
  END_STEP

  TRANSITION FROM Init TO Check
    := init;
  END_TRANSITION
  TRANSITION FROM Check TO Latch
    := set == 1;
  END_TRANSITION
  TRANSITION FROM Check TO Reset
    := reset == 1;
  END_TRANSITION
  TRANSITION FROM Check TO End
    := set == 0 and reset == 0;
  END_TRANSITION
  TRANSITION FROM Latch TO End
    := True;
  END_TRANSITION
  TRANSITION FROM Reset TO End
    := True;
  END_TRANSITION
END_PROGRAM

(* ---- 42_standard.st ---- *)
// Minimum of three

PROGRAM standard
  VAR
    a, b, c, min1, min2, init : INT;
  END_VAR

  ACTION act_Init
    min1 := a if a < b else b;
  END_ACTION

  ACTION act_Check
  END_ACTION

  ACTION act_Min2
    min2 := min1 if min1 < c else c;
  END_ACTION

  ACTION act_End
  END_ACTION

  INITIAL_STEP Init
    : act_Init(N);
  END_STEP

  STEP Check
    : act_Check(N);
  END_STEP

  STEP Min2
    : act_Min2(N);
  END_STEP

  STEP End
    : act_End(N);
  END_STEP

  TRANSITION FROM Init TO Check
    := init;
  END_TRANSITION
  TRANSITION FROM Check TO Min2
    := True;
  END_TRANSITION
  TRANSITION FROM Min2 TO End
    := True;
  END_TRANSITION
END_PROGRAM

(* ---- 42_upgraded.st ---- *)
// Minimum of three (Upgraded)

PROGRAM upgraded
  VAR
    a, b, c, min1, min2, init : INT;
  END_VAR

  ACTION act_Init
    min1 := min(a, b);
  END_ACTION

  ACTION act_Check
  END_ACTION

  ACTION act_Min2
    min2 := min(min1, c);
  END_ACTION

  ACTION act_End
  END_ACTION

  INITIAL_STEP Init
    : act_Init(N);
  END_STEP

  STEP Check
    : act_Check(N);
  END_STEP

  STEP Min2
    : act_Min2(N);
  END_STEP

  STEP End
    : act_End(N);
  END_STEP

  TRANSITION FROM Init TO Check
    := init;
  END_TRANSITION
  TRANSITION FROM Check TO Min2
    := True;
  END_TRANSITION
  TRANSITION FROM Min2 TO End
    := True;
  END_TRANSITION
END_PROGRAM

(* ---- 43_standard.st ---- *)
// Maximum of three

PROGRAM standard
  VAR
    a, b, c, max1, max2, init : INT;
  END_VAR

  ACTION act_Init
    max1 := a if a > b else b;
  END_ACTION

  ACTION act_Check
  END_ACTION

  ACTION act_Max2
    max2 := max1 if max1 > c else c;
  END_ACTION

  ACTION act_End
  END_ACTION

  INITIAL_STEP Init
    : act_Init(N);
  END_STEP

  STEP Check
    : act_Check(N);
  END_STEP

  STEP Max2
    : act_Max2(N);
  END_STEP

  STEP End
    : act_End(N);
  END_STEP

  TRANSITION FROM Init TO Check
    := init;
  END_TRANSITION
  TRANSITION FROM Check TO Max2
    := True;
  END_TRANSITION
  TRANSITION FROM Max2 TO End
    := True;
  END_TRANSITION
END_PROGRAM

(* ---- 43_upgraded.st ---- *)
// Maximum of three (Upgraded)

PROGRAM upgraded
  VAR
    a, b, c, max1, max2, init : INT;
  END_VAR

  ACTION act_Init
    max1 := max(a, b);
  END_ACTION

  ACTION act_Check
  END_ACTION

  ACTION act_Max2
    max2 := max(max1, c);
  END_ACTION

  ACTION act_End
  END_ACTION

  INITIAL_STEP Init
    : act_Init(N);
  END_STEP

  STEP Check
    : act_Check(N);
  END_STEP

  STEP Max2
    : act_Max2(N);
  END_STEP

  STEP End
    : act_End(N);
  END_STEP

  TRANSITION FROM Init TO Check
    := init;
  END_TRANSITION
  TRANSITION FROM Check TO Max2
    := True;
  END_TRANSITION
  TRANSITION FROM Max2 TO End
    := True;
  END_TRANSITION
END_PROGRAM

(* ---- 44_standard.st ---- *)
// Set value if condition

PROGRAM standard
  VAR
    cond, val, out, init : INT;
  END_VAR

  ACTION act_Init
    out := 0;
  END_ACTION

  ACTION act_Check
  END_ACTION

  ACTION act_Set
    out := val;
  END_ACTION

  ACTION act_End
  END_ACTION

  INITIAL_STEP Init
    : act_Init(N);
  END_STEP

  STEP Check
    : act_Check(N);
  END_STEP

  STEP Set
    : act_Set(N);
  END_STEP

  STEP End
    : act_End(N);
  END_STEP

  TRANSITION FROM Init TO Check
    := init;
  END_TRANSITION
  TRANSITION FROM Check TO Set
    := cond == 1;
  END_TRANSITION
  TRANSITION FROM Check TO End
    := cond == 0;
  END_TRANSITION
  TRANSITION FROM Set TO End
    := True;
  END_TRANSITION
END_PROGRAM

(* ---- 44_upgraded.st ---- *)
// Set value if condition (Upgraded)

PROGRAM upgraded
  VAR
    cond, val, out, init : INT;
  END_VAR

  ACTION act_Init
    out := 0;
  END_ACTION

  ACTION act_Check
  END_ACTION

  ACTION act_Set
    out := val * 2;
  END_ACTION

  ACTION act_End
  END_ACTION

  INITIAL_STEP Init
    : act_Init(N);
  END_STEP

  STEP Check
    : act_Check(N);
  END_STEP

  STEP Set
    : act_Set(N);
  END_STEP

  STEP End
    : act_End(N);
  END_STEP

  TRANSITION FROM Init TO Check
    := init;
  END_TRANSITION
  TRANSITION FROM Check TO Set
    := cond == 1;
  END_TRANSITION
  TRANSITION FROM Check TO End
    := cond == 0;
  END_TRANSITION
  TRANSITION FROM Set TO End
    := True;
  END_TRANSITION
END_PROGRAM

(* ---- 45_standard.st ---- *)
// Reset to default if condition

PROGRAM standard
  VAR
    cond, val, defval, out, init : INT;
  END_VAR

  ACTION act_Init
    out := val;
  END_ACTION

  ACTION act_Check
  END_ACTION

  ACTION act_Reset
    out := defval;
  END_ACTION

  ACTION act_End
  END_ACTION

  INITIAL_STEP Init
    : act_Init(N);
  END_STEP

  STEP Check
    : act_Check(N);
  END_STEP

  STEP Reset
    : act_Reset(N);
  END_STEP

  STEP End
    : act_End(N);
  END_STEP

  TRANSITION FROM Init TO Check
    := init;
  END_TRANSITION
  TRANSITION FROM Check TO Reset
    := cond == 1;
  END_TRANSITION
  TRANSITION FROM Check TO End
    := cond == 0;
  END_TRANSITION
  TRANSITION FROM Reset TO End
    := True;
  END_TRANSITION
END_PROGRAM

(* ---- 45_upgraded.st ---- *)
// Reset to default if condition (Upgraded)

PROGRAM upgraded
  VAR
    cond, val, defval, out, init : INT;
  END_VAR

  ACTION act_Init
    out := val + defval;
  END_ACTION

  ACTION act_Check
  END_ACTION

  ACTION act_Reset
    out := defval * 2;
  END_ACTION

  ACTION act_End
  END_ACTION

  INITIAL_STEP Init
    : act_Init(N);
  END_STEP

  STEP Check
    : act_Check(N);
  END_STEP

  STEP Reset
    : act_Reset(N);
  END_STEP

  STEP End
    : act_End(N);
  END_STEP

  TRANSITION FROM Init TO Check
    := init;
  END_TRANSITION
  TRANSITION FROM Check TO Reset
    := cond == 1;
  END_TRANSITION
  TRANSITION FROM Check TO End
    := cond == 0;
  END_TRANSITION
  TRANSITION FROM Reset TO End
    := True;
  END_TRANSITION
END_PROGRAM

(* ---- 46_standard.st ---- *)
// Sign Flip If Condition

PROGRAM standard
  VAR_INPUT
    input : INT;
  END_VAR
  VAR
    cond, out, init : INT;
  END_VAR

  ACTION act_Init
    out := input;
  END_ACTION

  ACTION act_Check
  END_ACTION

  ACTION act_Flip
    out := -input;
  END_ACTION

  ACTION act_End
  END_ACTION

  INITIAL_STEP Init
    : act_Init(N);
  END_STEP

  STEP Check
    : act_Check(N);
  END_STEP

  STEP Flip
    : act_Flip(N);
  END_STEP

  STEP End
    : act_End(N);
  END_STEP

  TRANSITION FROM Init TO Check
    := init;
  END_TRANSITION
  TRANSITION FROM Check TO Flip
    := cond == 1;
  END_TRANSITION
  TRANSITION FROM Check TO End
    := cond == 0;
  END_TRANSITION
  TRANSITION FROM Flip TO End
    := True;
  END_TRANSITION
END_PROGRAM

(* ---- 46_upgraded.st ---- *)
// Sign Flip If Condition (Upgraded)

PROGRAM upgraded
  VAR_INPUT
    input : INT;
  END_VAR
  VAR
    cond, out, init : INT;
  END_VAR

  ACTION act_Init
    out := input;
  END_ACTION

  ACTION act_Check
  END_ACTION

  ACTION act_Flip
    out := -input * 2;
  END_ACTION

  ACTION act_End
  END_ACTION

  INITIAL_STEP Init
    : act_Init(N);
  END_STEP

  STEP Check
    : act_Check(N);
  END_STEP

  STEP Flip
    : act_Flip(N);
  END_STEP

  STEP End
    : act_End(N);
  END_STEP

  TRANSITION FROM Init TO Check
    := init;
  END_TRANSITION
  TRANSITION FROM Check TO Flip
    := cond == 1;
  END_TRANSITION
  TRANSITION FROM Check TO End
    := cond == 0;
  END_TRANSITION
  TRANSITION FROM Flip TO End
    := True;
  END_TRANSITION
END_PROGRAM

(* ---- 47_standard.st ---- *)
// Reset If Negative

PROGRAM standard
  VAR_INPUT
    input : INT;
  END_VAR
  VAR
    out, init : INT;
  END_VAR

  ACTION act_Init
    out := input;
  END_ACTION

  ACTION act_Check
  END_ACTION

  ACTION act_Reset
    out := 0;
  END_ACTION

  ACTION act_End
  END_ACTION

  INITIAL_STEP Init
    : act_Init(N);
  END_STEP

  STEP Check
    : act_Check(N);
  END_STEP

  STEP Reset
    : act_Reset(N);
  END_STEP

  STEP End
    : act_End(N);
  END_STEP

  TRANSITION FROM Init TO Check
    := init;
  END_TRANSITION
  TRANSITION FROM Check TO Reset
    := input < 0;
  END_TRANSITION
  TRANSITION FROM Check TO End
    := input >= 0;
  END_TRANSITION
  TRANSITION FROM Reset TO End
    := True;
  END_TRANSITION
END_PROGRAM

(* ---- 47_upgraded.st ---- *)
// Reset If Negative (Upgraded)

PROGRAM upgraded
  VAR_INPUT
    input : INT;
  END_VAR
  VAR
    out, init : INT;
  END_VAR

  ACTION act_Init
    out := input * 2;
  END_ACTION

  ACTION act_Check
  END_ACTION

  ACTION act_Reset
    out := input + 1;
  END_ACTION

  ACTION act_End
  END_ACTION

  INITIAL_STEP Init
    : act_Init(N);
  END_STEP

  STEP Check
    : act_Check(N);
  END_STEP

  STEP Reset
    : act_Reset(N);
  END_STEP

  STEP End
    : act_End(N);
  END_STEP

  TRANSITION FROM Init TO Check
    := init;
  END_TRANSITION
  TRANSITION FROM Check TO Reset
    := input < 0;
  END_TRANSITION
  TRANSITION FROM Check TO End
    := input >= 0;
  END_TRANSITION
  TRANSITION FROM Reset TO End
    := True;
  END_TRANSITION
END_PROGRAM

(* ---- 48_standard.st ---- *)
// Set to Max if Exceeds

PROGRAM standard
  VAR_INPUT
    input : INT;
  END_VAR
  VAR
    maxval, out, init : INT;
  END_VAR

  ACTION act_Init
    out := input;
  END_ACTION

  ACTION act_Check
  END_ACTION

  ACTION act_SetMax
    out := maxval;
  END_ACTION

  ACTION act_End
  END_ACTION

  INITIAL_STEP Init
    : act_Init(N);
  END_STEP

  STEP Check
    : act_Check(N);
  END_STEP

  STEP SetMax
    : act_SetMax(N);
  END_STEP

  STEP End
    : act_End(N);
  END_STEP

  TRANSITION FROM Init TO Check
    := init;
  END_TRANSITION
  TRANSITION FROM Check TO SetMax
    := input > maxval;
  END_TRANSITION
  TRANSITION FROM Check TO End
    := input <= maxval;
  END_TRANSITION
  TRANSITION FROM SetMax TO End
    := True;
  END_TRANSITION
END_PROGRAM

(* ---- 48_upgraded.st ---- *)
// Set to Max if Exceeds (Upgraded)

PROGRAM upgraded
  VAR_INPUT
    input : INT;
  END_VAR
  VAR
    maxval, out, init : INT;
  END_VAR

  ACTION act_Init
    out := input;
  END_ACTION

  ACTION act_Check
  END_ACTION

  ACTION act_SetMax
    out := maxval * 2;
  END_ACTION

  ACTION act_End
  END_ACTION

  INITIAL_STEP Init
    : act_Init(N);
  END_STEP

  STEP Check
    : act_Check(N);
  END_STEP

  STEP SetMax
    : act_SetMax(N);
  END_STEP

  STEP End
    : act_End(N);
  END_STEP

  TRANSITION FROM Init TO Check
    := init;
  END_TRANSITION
  TRANSITION FROM Check TO SetMax
    := input > maxval;
  END_TRANSITION
  TRANSITION FROM Check TO End
    := input <= maxval;
  END_TRANSITION
  TRANSITION FROM SetMax TO End
    := True;
  END_TRANSITION
END_PROGRAM

(* ---- 49_standard.st ---- *)
// Set to Min if Below

PROGRAM standard
  VAR_INPUT
    input : INT;
  END_VAR
  VAR
    minval, out, init : INT;
  END_VAR

  ACTION act_Init
    out := input;
  END_ACTION

  ACTION act_Check
  END_ACTION

  ACTION act_SetMin
    out := minval;
  END_ACTION

  ACTION act_End
  END_ACTION

  INITIAL_STEP Init
    : act_Init(N);
  END_STEP

  STEP Check
    : act_Check(N);
  END_STEP

  STEP SetMin
    : act_SetMin(N);
  END_STEP

  STEP End
    : act_End(N);
  END_STEP

  TRANSITION FROM Init TO Check
    := init;
  END_TRANSITION
  TRANSITION FROM Check TO SetMin
    := input < minval;
  END_TRANSITION
  TRANSITION FROM Check TO End
    := input >= minval;
  END_TRANSITION
  TRANSITION FROM SetMin TO End
    := True;
  END_TRANSITION
END_PROGRAM

(* ---- 49_upgraded.st ---- *)
// Set to Min if Below (Upgraded)

PROGRAM upgraded
  VAR_INPUT
    input : INT;
  END_VAR
  VAR
    minval, out, init : INT;
  END_VAR

  ACTION act_Init
    out := input;
  END_ACTION

  ACTION act_Check
  END_ACTION

  ACTION act_SetMin
    out := minval - 1;
  END_ACTION

  ACTION act_End
  END_ACTION

  INITIAL_STEP Init
    : act_Init(N);
  END_STEP

  STEP Check
    : act_Check(N);
  END_STEP

  STEP SetMin
    : act_SetMin(N);
  END_STEP

  STEP End
    : act_End(N);
  END_STEP

  TRANSITION FROM Init TO Check
    := init;
  END_TRANSITION
  TRANSITION FROM Check TO SetMin
    := input < minval;
  END_TRANSITION
  TRANSITION FROM Check TO End
    := input >= minval;
  END_TRANSITION
  TRANSITION FROM SetMin TO End
    := True;
  END_TRANSITION
END_PROGRAM

(* ---- 4_standard.st ---- *)
// Delay On Timer

PROGRAM standard
  VAR_INPUT
    input : INT;
  END_VAR
  VAR_OUTPUT
    output : INT;
  END_VAR
  VAR
    timer, delay, init : INT;
  END_VAR

  ACTION act_Init
    timer := 0; output := 0;
  END_ACTION

  ACTION act_Check
  END_ACTION

  ACTION act_Count
    timer := timer + 1;
  END_ACTION

  ACTION act_On
    output := 1;
  END_ACTION

  ACTION act_Reset
    timer := 0; output := 0;
  END_ACTION

  ACTION act_End
  END_ACTION

  INITIAL_STEP Init
    : act_Init(N);
  END_STEP

  STEP Check
    : act_Check(N);
  END_STEP

  STEP Count
    : act_Count(N);
  END_STEP

  STEP On
    : act_On(N);
  END_STEP

  STEP Reset
    : act_Reset(N);
  END_STEP

  STEP End
    : act_End(N);
  END_STEP

  TRANSITION FROM Init TO Check
    := init;
  END_TRANSITION
  TRANSITION FROM Check TO Count
    := input == 1 and timer < delay;
  END_TRANSITION
  TRANSITION FROM Count TO Check
    := True;
  END_TRANSITION
  TRANSITION FROM Check TO On
    := input == 1 and timer >= delay;
  END_TRANSITION
  TRANSITION FROM On TO Check
    := True;
  END_TRANSITION
  TRANSITION FROM Check TO Reset
    := input == 0;
  END_TRANSITION
  TRANSITION FROM Reset TO Check
    := True;
  END_TRANSITION
END_PROGRAM

(* ---- 4_upgraded.st ---- *)
// Delay On Timer (Upgraded)

PROGRAM upgraded
  VAR_INPUT
    input : INT;
  END_VAR
  VAR_OUTPUT
    output : INT;
  END_VAR
  VAR
    timer, delay, step, scale, init : INT;
  END_VAR

  ACTION act_Init
    timer := 0; output := 0;
  END_ACTION

  ACTION act_Check
  END_ACTION

  ACTION act_Count
    timer := timer + step;
  END_ACTION

  ACTION act_On
    output := timer * scale;
  END_ACTION

  ACTION act_Reset
    timer := 0; output := 0;
  END_ACTION

  ACTION act_End
  END_ACTION

  INITIAL_STEP Init
    : act_Init(N);
  END_STEP

  STEP Check
    : act_Check(N);
  END_STEP

  STEP Count
    : act_Count(N);
  END_STEP

  STEP On
    : act_On(N);
  END_STEP

  STEP Reset
    : act_Reset(N);
  END_STEP

  STEP End
    : act_End(N);
  END_STEP

  TRANSITION FROM Init TO Check
    := init;
  END_TRANSITION
  TRANSITION FROM Check TO Count
    := input == 1 and timer < delay;
  END_TRANSITION
  TRANSITION FROM Count TO Check
    := True;
  END_TRANSITION
  TRANSITION FROM Check TO On
    := input == 1 and timer >= delay;
  END_TRANSITION
  TRANSITION FROM On TO Check
    := True;
  END_TRANSITION
  TRANSITION FROM Check TO Reset
    := input == 0;
  END_TRANSITION
  TRANSITION FROM Reset TO Check
    := True;
  END_TRANSITION
END_PROGRAM

(* ---- 50_standard.st ---- *)
// Reset If Out Of Bounds

PROGRAM standard
  VAR_INPUT
    input : INT;
  END_VAR
  VAR
    minval, maxval, out, init : INT;
  END_VAR

  ACTION act_Init
    out := input;
  END_ACTION

  ACTION act_Check
  END_ACTION

  ACTION act_Reset
    out := 0;
  END_ACTION

  ACTION act_End
  END_ACTION

  INITIAL_STEP Init
    : act_Init(N);
  END_STEP

  STEP Check
    : act_Check(N);
  END_STEP

  STEP Reset
    : act_Reset(N);
  END_STEP

  STEP End
    : act_End(N);
  END_STEP

  TRANSITION FROM Init TO Check
    := init;
  END_TRANSITION
  TRANSITION FROM Check TO Reset
    := input < minval or input > maxval;
  END_TRANSITION
  TRANSITION FROM Check TO End
    := input >= minval and input <= maxval;
  END_TRANSITION
  TRANSITION FROM Reset TO End
    := True;
  END_TRANSITION
END_PROGRAM

(* ---- 50_upgraded.st ---- *)
// Reset If Out Of Bounds (Upgraded)

PROGRAM upgraded
  VAR_INPUT
    input : INT;
  END_VAR
  VAR
    minval, maxval, out, init : INT;
  END_VAR

  ACTION act_Init
    out := input * 2;
  END_ACTION

  ACTION act_Check
  END_ACTION

  ACTION act_Reset
    out := input + maxval;
  END_ACTION

  ACTION act_End
  END_ACTION

  INITIAL_STEP Init
    : act_Init(N);
  END_STEP

  STEP Check
    : act_Check(N);
  END_STEP

  STEP Reset
    : act_Reset(N);
  END_STEP

  STEP End
    : act_End(N);
  END_STEP

  TRANSITION FROM Init TO Check
    := init;
  END_TRANSITION
  TRANSITION FROM Check TO Reset
    := input < minval or input > maxval;
  END_TRANSITION
  TRANSITION FROM Check TO End
    := input >= minval and input <= maxval;
  END_TRANSITION
  TRANSITION FROM Reset TO End
    := True;
  END_TRANSITION
END_PROGRAM

(* ---- 5_standard.st ---- *)
// Delay Off Timer

PROGRAM standard
  VAR_INPUT
    input : INT;
  END_VAR
  VAR_OUTPUT
    output : INT;
  END_VAR
  VAR
    timer, delay, init : INT;
  END_VAR

  ACTION act_Init
    timer := 0; output := 0;
  END_ACTION

  ACTION act_Check
  END_ACTION

  ACTION act_Set
    output := 1;
  END_ACTION

  ACTION act_Count
    timer := timer + 1;
  END_ACTION

  ACTION act_Reset
    timer := 0; output := 0;
  END_ACTION

  ACTION act_End
  END_ACTION

  INITIAL_STEP Init
    : act_Init(N);
  END_STEP

  STEP Check
    : act_Check(N);
  END_STEP

  STEP Set
    : act_Set(N);
  END_STEP

  STEP Count
    : act_Count(N);
  END_STEP

  STEP Reset
    : act_Reset(N);
  END_STEP

  STEP End
    : act_End(N);
  END_STEP

  TRANSITION FROM Init TO Check
    := init;
  END_TRANSITION
  TRANSITION FROM Check TO Set
    := input == 1;
  END_TRANSITION
  TRANSITION FROM Set TO Check
    := True;
  END_TRANSITION
  TRANSITION FROM Check TO Count
    := input == 0 and timer < delay;
  END_TRANSITION
  TRANSITION FROM Count TO Check
    := True;
  END_TRANSITION
  TRANSITION FROM Check TO Reset
    := input == 0 and timer >= delay;
  END_TRANSITION
  TRANSITION FROM Reset TO Check
    := True;
  END_TRANSITION
END_PROGRAM

(* ---- 5_upgraded.st ---- *)
// Delay Off Timer (Upgraded)

PROGRAM upgraded
  VAR_INPUT
    input : INT;
  END_VAR
  VAR_OUTPUT
    output : INT;
  END_VAR
  VAR
    timer, delay, init : INT;
  END_VAR

  ACTION act_Init
    timer := 0; output := 0;
  END_ACTION

  ACTION act_Check
  END_ACTION

  ACTION act_Set
    output := timer + 1;
  END_ACTION

  ACTION act_Count
    timer := timer + 2;
  END_ACTION

  ACTION act_Reset
    timer := 0; output := 0;
  END_ACTION

  ACTION act_End
  END_ACTION

  INITIAL_STEP Init
    : act_Init(N);
  END_STEP

  STEP Check
    : act_Check(N);
  END_STEP

  STEP Set
    : act_Set(N);
  END_STEP

  STEP Count
    : act_Count(N);
  END_STEP

  STEP Reset
    : act_Reset(N);
  END_STEP

  STEP End
    : act_End(N);
  END_STEP

  TRANSITION FROM Init TO Check
    := init;
  END_TRANSITION
  TRANSITION FROM Check TO Set
    := input == 1;
  END_TRANSITION
  TRANSITION FROM Set TO Check
    := True;
  END_TRANSITION
  TRANSITION FROM Check TO Count
    := input == 0 and timer < delay;
  END_TRANSITION
  TRANSITION FROM Count TO Check
    := True;
  END_TRANSITION
  TRANSITION FROM Check TO Reset
    := input == 0 and timer >= delay;
  END_TRANSITION
  TRANSITION FROM Reset TO Check
    := True;
  END_TRANSITION
END_PROGRAM

(* ---- 6_standard.st ---- *)
// Rising Edge Detection

PROGRAM standard
  VAR_INPUT
    input : INT;
  END_VAR
  VAR
    last, edge, init : INT;
  END_VAR

  ACTION act_Init
    last := 0; edge := 0;
  END_ACTION

  ACTION act_Check
  END_ACTION

  ACTION act_Detect
    edge := 1;
  END_ACTION

  ACTION act_End
    last := input; edge := 0;
  END_ACTION

  INITIAL_STEP Init
    : act_Init(N);
  END_STEP

  STEP Check
    : act_Check(N);
  END_STEP

  STEP Detect
    : act_Detect(N);
  END_STEP

  STEP End
    : act_End(N);
  END_STEP

  TRANSITION FROM Init TO Check
    := init;
  END_TRANSITION
  TRANSITION FROM Check TO Detect
    := input == 1 and last == 0;
  END_TRANSITION
  TRANSITION FROM Detect TO End
    := True;
  END_TRANSITION
  TRANSITION FROM Check TO End
    := input == 0 or last == 1;
  END_TRANSITION
END_PROGRAM

(* ---- 6_upgraded.st ---- *)
// Rising Edge Detection (Upgraded)

PROGRAM upgraded
  VAR_INPUT
    input : INT;
  END_VAR
  VAR
    last, edge, edge_count, init : INT;
  END_VAR

  ACTION act_Init
    last := 0; edge := 0; edge_count := 0;
  END_ACTION

  ACTION act_Check
  END_ACTION

  ACTION act_Detect
    edge := 1; edge_count := edge_count + 1;
  END_ACTION

  ACTION act_End
    last := input; edge := 0;
  END_ACTION

  INITIAL_STEP Init
    : act_Init(N);
  END_STEP

  STEP Check
    : act_Check(N);
  END_STEP

  STEP Detect
    : act_Detect(N);
  END_STEP

  STEP End
    : act_End(N);
  END_STEP

  TRANSITION FROM Init TO Check
    := init;
  END_TRANSITION
  TRANSITION FROM Check TO Detect
    := input == 1 and last == 0;
  END_TRANSITION
  TRANSITION FROM Detect TO End
    := True;
  END_TRANSITION
  TRANSITION FROM Check TO End
    := input == 0 or last == 1;
  END_TRANSITION
END_PROGRAM

(* ---- 7_standard.st ---- *)
// Falling Edge Detection

PROGRAM standard
  VAR_INPUT
    input : INT;
  END_VAR
  VAR
    last, edge, init : INT;
  END_VAR

  ACTION act_Init
    last := 1; edge := 0;
  END_ACTION

  ACTION act_Check
  END_ACTION

  ACTION act_Detect
    edge := 1;
  END_ACTION

  ACTION act_End
    last := input; edge := 0;
  END_ACTION

  INITIAL_STEP Init
    : act_Init(N);
  END_STEP

  STEP Check
    : act_Check(N);
  END_STEP

  STEP Detect
    : act_Detect(N);
  END_STEP

  STEP End
    : act_End(N);
  END_STEP

  TRANSITION FROM Init TO Check
    := init;
  END_TRANSITION
  TRANSITION FROM Check TO Detect
    := input == 0 and last == 1;
  END_TRANSITION
  TRANSITION FROM Detect TO End
    := True;
  END_TRANSITION
  TRANSITION FROM Check TO End
    := input == 1 or last == 0;
  END_TRANSITION
END_PROGRAM

(* ---- 7_upgraded.st ---- *)
// Falling Edge Detection (Upgraded)

PROGRAM upgraded
  VAR_INPUT
    input : INT;
  END_VAR
  VAR
    last, edge, edge_count, init : INT;
  END_VAR

  ACTION act_Init
    last := 1; edge := 0; edge_count := 0;
  END_ACTION

  ACTION act_Check
  END_ACTION

  ACTION act_Detect
    edge := 1; edge_count := edge_count + 1;
  END_ACTION

  ACTION act_End
    last := input; edge := 0;
  END_ACTION

  INITIAL_STEP Init
    : act_Init(N);
  END_STEP

  STEP Check
    : act_Check(N);
  END_STEP

  STEP Detect
    : act_Detect(N);
  END_STEP

  STEP End
    : act_End(N);
  END_STEP

  TRANSITION FROM Init TO Check
    := init;
  END_TRANSITION
  TRANSITION FROM Check TO Detect
    := input == 0 and last == 1;
  END_TRANSITION
  TRANSITION FROM Detect TO End
    := True;
  END_TRANSITION
  TRANSITION FROM Check TO End
    := input == 1 or last == 0;
  END_TRANSITION
END_PROGRAM

(* ---- 8_standard.st ---- *)
// Pulse Generator (fixed width)

PROGRAM standard
  VAR
    trigger, timer, width, pulse, init : INT;
  END_VAR

  ACTION act_Init
    timer := 0; pulse := 0;
  END_ACTION

  ACTION act_Check
  END_ACTION

  ACTION act_StartPulse
    pulse := 1; timer := 1;
  END_ACTION

  ACTION act_Pulse
    timer := timer + 1;
  END_ACTION

  ACTION act_StopPulse
    pulse := 0; timer := 0;
  END_ACTION

  ACTION act_End
  END_ACTION

  INITIAL_STEP Init
    : act_Init(N);
  END_STEP

  STEP Check
    : act_Check(N);
  END_STEP

  STEP StartPulse
    : act_StartPulse(N);
  END_STEP

  STEP Pulse
    : act_Pulse(N);
  END_STEP

  STEP StopPulse
    : act_StopPulse(N);
  END_STEP

  STEP End
    : act_End(N);
  END_STEP

  TRANSITION FROM Init TO Check
    := init;
  END_TRANSITION
  TRANSITION FROM Check TO StartPulse
    := trigger == 1;
  END_TRANSITION
  TRANSITION FROM StartPulse TO Pulse
    := True;
  END_TRANSITION
  TRANSITION FROM Pulse TO Pulse
    := timer < width;
  END_TRANSITION
  TRANSITION FROM Pulse TO StopPulse
    := timer >= width;
  END_TRANSITION
  TRANSITION FROM StopPulse TO Check
    := True;
  END_TRANSITION
END_PROGRAM

(* ---- 8_upgraded.st ---- *)
// Pulse Generator (fixed width) (Upgraded)

PROGRAM upgraded
  VAR
    trigger, timer, width, pulse, init : INT;
  END_VAR

  ACTION act_Init
    timer := 0; pulse := 0;
  END_ACTION

  ACTION act_Check
  END_ACTION

  ACTION act_StartPulse
    pulse := 1; timer := 1;
  END_ACTION

  ACTION act_Pulse
    timer := timer * 2;
  END_ACTION

  ACTION act_StopPulse
    pulse := 0; timer := 0;
  END_ACTION

  ACTION act_End
  END_ACTION

  INITIAL_STEP Init
    : act_Init(N);
  END_STEP

  STEP Check
    : act_Check(N);
  END_STEP

  STEP StartPulse
    : act_StartPulse(N);
  END_STEP

  STEP Pulse
    : act_Pulse(N);
  END_STEP

  STEP StopPulse
    : act_StopPulse(N);
  END_STEP

  STEP End
    : act_End(N);
  END_STEP

  TRANSITION FROM Init TO Check
    := init;
  END_TRANSITION
  TRANSITION FROM Check TO StartPulse
    := trigger == 1;
  END_TRANSITION
  TRANSITION FROM StartPulse TO Pulse
    := True;
  END_TRANSITION
  TRANSITION FROM Pulse TO Pulse
    := timer < width;
  END_TRANSITION
  TRANSITION FROM Pulse TO StopPulse
    := timer >= width;
  END_TRANSITION
  TRANSITION FROM StopPulse TO Check
    := True;
  END_TRANSITION
END_PROGRAM

(* ---- 9_standard.st ---- *)
// Up Counter

PROGRAM standard
  VAR_INPUT
    input : INT;
  END_VAR
  VAR
    reset, cnt, max, init : INT;
  END_VAR

  ACTION act_Init
    cnt := 0;
  END_ACTION

  ACTION act_Check
  END_ACTION

  ACTION act_Count
    cnt := cnt + 1;
  END_ACTION

  ACTION act_Reset
    cnt := 0;
  END_ACTION

  ACTION act_End
  END_ACTION

  INITIAL_STEP Init
    : act_Init(N);
  END_STEP

  STEP Check
    : act_Check(N);
  END_STEP

  STEP Count
    : act_Count(N);
  END_STEP

  STEP Reset
    : act_Reset(N);
  END_STEP

  STEP End
    : act_End(N);
  END_STEP

  TRANSITION FROM Init TO Check
    := init;
  END_TRANSITION
  TRANSITION FROM Check TO Count
    := input == 1 and cnt < max;
  END_TRANSITION
  TRANSITION FROM Count TO Check
    := True;
  END_TRANSITION
  TRANSITION FROM Check TO Reset
    := reset == 1;
  END_TRANSITION
  TRANSITION FROM Reset TO Check
    := True;
  END_TRANSITION
END_PROGRAM

(* ---- 9_upgraded.st ---- *)
// Up Counter (Upgraded)

PROGRAM upgraded
  VAR_INPUT
    input : INT;
  END_VAR
  VAR
    reset, cnt, max, init : INT;
  END_VAR

  ACTION act_Init
    cnt := 0;
  END_ACTION

  ACTION act_Check
  END_ACTION

  ACTION act_Count
    cnt := cnt + 2;
  END_ACTION

  ACTION act_Reset
    cnt := 0;
  END_ACTION

  ACTION act_End
  END_ACTION

  INITIAL_STEP Init
    : act_Init(N);
  END_STEP

  STEP Check
    : act_Check(N);
  END_STEP

  STEP Count
    : act_Count(N);
  END_STEP

  STEP Reset
    : act_Reset(N);
  END_STEP

  STEP End
    : act_End(N);
  END_STEP

  TRANSITION FROM Init TO Check
    := init;
  END_TRANSITION
  TRANSITION FROM Check TO Count
    := input == 1 and cnt < max;
  END_TRANSITION
  TRANSITION FROM Count TO Check
    := True;
  END_TRANSITION
  TRANSITION FROM Check TO Reset
    := reset == 1;
  END_TRANSITION
  TRANSITION FROM Reset TO Check
    := True;
  END_TRANSITION
END_PROGRAM
